LIN {X 0,Y 411.31,Z 349.876,A -85,B 0,C 180,E1 -10435.099,E2 -10435.099} C_VEL
LIN {X 0,Y 411.512,Z 349.85,A -85,B 0,C 180,E1 -10438.042,E2 -10438.042} C_VEL
LIN {X 0,Y 411.64,Z 349.837,A -85,B 0,C 180,E1 -10440,E2 -10440} C_VEL
LIN {X 0,Y 411.465,Z 349.857,A -85,B 0,C 180,E1 -10442.937,E2 -10442.937} C_VEL
LIN {X 0,Y 411.458,Z 349.857,A -85,B 0,C 180,E1 -10446.867,E2 -10446.867} C_VEL
LIN {X 0,Y 411.292,Z 349.877,A -85,B 0,C 180,E1 -10449.839,E2 -10449.839} C_VEL
LIN {X 0,Y 411.303,Z 349.874,A -85,B 0,C 180,E1 -10453.104,E2 -10453.104} C_VEL
LIN {X 0,Y 411.26,Z 349.883,A -85,B 0,C 180,E1 -10456.869,E2 -10456.869} C_VEL
LIN {X 0,Y 411.228,Z 349.888,A -85,B 0,C 180,E1 -10459.987,E2 -10459.987} C_VEL
LIN {X 0,Y 411.201,Z 349.893,A -85,B 0,C 180,E1 -10463.148,E2 -10463.148} C_VEL
LIN {X 0,Y 411.235,Z 349.889,A -85,B 0,C 180,E1 -10466.381,E2 -10466.381} C_VEL
LIN {X 0,Y 411.209,Z 349.89,A -85,B 0,C 180,E1 -10469.712,E2 -10469.712} C_VEL
LIN {X 0,Y 411.204,Z 349.89,A -85,B 0,C 180,E1 -10473.156,E2 -10473.156} C_VEL
LIN {X 0,Y 411.193,Z 349.891,A -85,B 0,C 180,E1 -10476.553,E2 -10476.553} C_VEL
LIN {X 0,Y 411.247,Z 349.991,A -85,B 0,C 180,E1 -10479.561,E2 -10479.561} C_VEL
LIN {X 0,Y 412.074,Z 354.924,A -85,B 0,C 180,E1 -10483.016,E2 -10483.016} C_VEL
LIN {X 0,Y 412.925,Z 360.046,A -85,B 0,C 180,E1 -10486.331,E2 -10486.331} C_VEL
LIN {X 0,Y 413.217,Z 363.579,A -85,B 0,C 180,E1 -10488.448,E2 -10488.448} C_VEL
LIN {X 0,Y 412.818,Z 369.165,A -85,B 0,C 180,E1 -10491.547,E2 -10491.547} C_VEL
LIN {X 0,Y 412.354,Z 375.474,A -85,B 0,C 180,E1 -10494.894,E2 -10494.894} C_VEL
LIN {X 0,Y 411.903,Z 382.668,A -85,B 0,C 180,E1 -10498.552,E2 -10498.552} C_VEL
LIN {X 0,Y 411.323,Z 389.578,A -85,B 0,C 180,E1 -10501.974,E2 -10501.974} C_VEL
LIN {X 0,Y 410.999,Z 395.754,A -85,B 0,C 180,E1 -10505.028,E2 -10505.028} C_VEL
LIN {X 0,Y 415.661,Z 413.767,A -85,B 0,C 180,E1 -10505.779,E2 -10505.779} C_VEL
LIN {X 0,Y 418.601,Z 427.932,A -85,B 0,C 180,E1 -10506.506,E2 -10506.506} C_VEL
LIN {X 0,Y 419.89,Z 436.709,A -85,B 0,C 180,E1 -10507.01,E2 -10507.01} C_VEL
LIN {X 0,Y 418.871,Z 450.945,A -85,B 0,C 180,E1 -10507.821,E2 -10507.821} C_VEL
LIN {X 0,Y 417.535,Z 464.473,A -85,B 0,C 180,E1 -10508.784,E2 -10508.784} C_VEL
LIN {X 0,Y 416.15,Z 478.262,A -85,B 0,C 180,E1 -10510.003,E2 -10510.003} C_VEL
LIN {X 0,Y 414.83,Z 490.734,A -85,B 0,C 180,E1 -10511.349,E2 -10511.349} C_VEL
LIN {X 0,Y 413.539,Z 503.017,A -85,B 0,C 180,E1 -10512.953,E2 -10512.953} C_VEL
LIN {X 0,Y 412.356,Z 513.929,A -85,B 0,C 180,E1 -10514.683,E2 -10514.683} C_VEL
LIN {X 0,Y 411.484,Z 523.109,A -85,B 0,C 180,E1 -10516.435,E2 -10516.435} C_VEL
LIN {X 0,Y 410.878,Z 530.585,A -85,B 0,C 180,E1 -10518.156,E2 -10518.156} C_VEL
LIN {X 0,Y 410.341,Z 537.64,A -85,B 0,C 180,E1 -10520.139,E2 -10520.139} C_VEL
LIN {X 0,Y 410.152,Z 543.2,A -85,B 0,C 180,E1 -10522.121,E2 -10522.121} C_VEL
LIN {X 0,Y 409.988,Z 547.402,A -85,B 0,C 180,E1 -10524.097,E2 -10524.097} C_VEL
LIN {X 0,Y 409.933,Z 550.351,A -85,B 0,C 180,E1 -10526.068,E2 -10526.068} C_VEL
LIN {X 0,Y 410.009,Z 552.115,A -85,B 0,C 180,E1 -10528.036,E2 -10528.036} C_VEL
LIN {X 0,Y 409.968,Z 552.715,A -85,B 0,C 180,E1 -10530,E2 -10530} C_VEL
LIN {X 0,Y 410.009,Z 552.11,A -85,B 0,C 180,E1 -10531.965,E2 -10531.965} C_VEL
LIN {X 0,Y 409.936,Z 550.342,A -85,B 0,C 180,E1 -10533.933,E2 -10533.933} C_VEL
LIN {X 0,Y 410.034,Z 547.395,A -85,B 0,C 180,E1 -10535.903,E2 -10535.903} C_VEL
LIN {X 0,Y 410.153,Z 543.193,A -85,B 0,C 180,E1 -10537.879,E2 -10537.879} C_VEL
LIN {X 0,Y 410.341,Z 537.627,A -85,B 0,C 180,E1 -10539.862,E2 -10539.862} C_VEL
LIN {X 0,Y 410.884,Z 530.561,A -85,B 0,C 180,E1 -10541.845,E2 -10541.845} C_VEL
LIN {X 0,Y 411.591,Z 521.772,A -85,B 0,C 180,E1 -10543.831,E2 -10543.831} C_VEL
LIN {X 0,Y 412.495,Z 512.449,A -85,B 0,C 180,E1 -10545.566,E2 -10545.566} C_VEL
LIN {X 0,Y 413.491,Z 502.979,A -85,B 0,C 180,E1 -10547.05,E2 -10547.05} C_VEL
LIN {X 0,Y 414.8,Z 491.133,A -85,B 0,C 180,E1 -10548.601,E2 -10548.601} C_VEL
LIN {X 0,Y 416.041,Z 479.441,A -85,B 0,C 180,E1 -10549.875,E2 -10549.875} C_VEL
LIN {X 0,Y 417.365,Z 465.924,A -85,B 0,C 180,E1 -10551.097,E2 -10551.097} C_VEL
LIN {X 0,Y 418.711,Z 452.668,A -85,B 0,C 180,E1 -10552.059,E2 -10552.059} C_VEL
LIN {X 0,Y 419.657,Z 439.382,A -85,B 0,C 180,E1 -10552.846,E2 -10552.846} C_VEL
LIN {X 0,Y 419.836,Z 435.502,A -85,B 0,C 180,E1 -10553.05,E2 -10553.05} C_VEL
LIN {X 0,Y 417.05,Z 420.044,A -85,B 0,C 180,E1 -10553.907,E2 -10553.907} C_VEL
LIN {X 0,Y 413.473,Z 405.19,A -85,B 0,C 180,E1 -10554.597,E2 -10554.597} C_VEL
LIN {X 0,Y 410.984,Z 395.734,A -85,B 0,C 180,E1 -10554.976,E2 -10554.976} C_VEL
LIN {X 0,Y 411.42,Z 388.428,A -85,B 0,C 180,E1 -10558.575,E2 -10558.575} C_VEL
LIN {X 0,Y 411.784,Z 382.677,A -85,B 0,C 180,E1 -10561.421,E2 -10561.421} C_VEL
LIN {X 0,Y 412.245,Z 377.131,A -85,B 0,C 180,E1 -10564.235,E2 -10564.235} C_VEL
LIN {X 0,Y 412.687,Z 370.278,A -85,B 0,C 180,E1 -10567.813,E2 -10567.813} C_VEL
LIN {X 0,Y 413.181,Z 364.609,A -85,B 0,C 180,E1 -10570.91,E2 -10570.91} C_VEL
LIN {X 0,Y 413.04,Z 361.111,A -85,B 0,C 180,E1 -10572.975,E2 -10572.975} C_VEL
LIN {X 0,Y 412.407,Z 356.805,A -85,B 0,C 180,E1 -10575.704,E2 -10575.704} C_VEL
LIN {X 0,Y 411.632,Z 352.375,A -85,B 0,C 180,E1 -10578.698,E2 -10578.698} C_VEL
LIN {X 0,Y 411.232,Z 349.887,A -85,B 0,C 180,E1 -10580.521,E2 -10580.521} C_VEL
LIN {X 0,Y 411.198,Z 349.896,A -85,B 0,C 180,E1 -10583.447,E2 -10583.447} C_VEL
LIN {X 0,Y 411.209,Z 349.891,A -85,B 0,C 180,E1 -10586.874,E2 -10586.874} C_VEL
LIN {X 0,Y 411.235,Z 349.888,A -85,B 0,C 180,E1 -10590.644,E2 -10590.644} C_VEL
LIN {X 0,Y 411.24,Z 349.887,A -85,B 0,C 180,E1 -10593.619,E2 -10593.619} C_VEL
LIN {X 0,Y 411.206,Z 349.892,A -85,B 0,C 180,E1 -10596.853,E2 -10596.853} C_VEL
LIN {X 0,Y 411.218,Z 349.89,A -85,B 0,C 180,E1 -10600.05,E2 -10600.05} C_VEL
LIN {X 0,Y 411.266,Z 349.885,A -85,B 0,C 180,E1 -10603.131,E2 -10603.131} C_VEL
LIN {X 0,Y 411.309,Z 349.878,A -85,B 0,C 180,E1 -10606.896,E2 -10606.896} C_VEL
LIN {X 0,Y 411.296,Z 349.879,A -85,B 0,C 180,E1 -10610.161,E2 -10610.161} C_VEL
LIN {X 0,Y 411.464,Z 349.857,A -85,B 0,C 180,E1 -10613.133,E2 -10613.133} C_VEL
LIN {X 0,Y 411.314,Z 349.878,A -85,B 0,C 180,E1 -10615.099,E2 -10615.099} C_VEL
LIN {X 0,Y 411.517,Z 349.851,A -85,B 0,C 180,E1 -10618.043,E2 -10618.043} C_VEL
LIN {X 0,Y 411.644,Z 349.834,A -85,B 0,C 180,E1 -10620,E2 -10620} C_VEL
LIN {X 0,Y 411.468,Z 349.855,A -85,B 0,C 180,E1 -10622.937,E2 -10622.937} C_VEL
LIN {X 0,Y 411.464,Z 349.853,A -85,B 0,C 180,E1 -10626.867,E2 -10626.867} C_VEL
LIN {X 0,Y 411.297,Z 349.876,A -85,B 0,C 180,E1 -10629.839,E2 -10629.839} C_VEL
LIN {X 0,Y 411.309,Z 349.855,A -85,B 0,C 180,E1 -10633.104,E2 -10633.104} C_VEL
LIN {X 0,Y 411.266,Z 349.881,A -85,B 0,C 180,E1 -10636.869,E2 -10636.869} C_VEL
LIN {X 0,Y 411.234,Z 349.867,A -85,B 0,C 180,E1 -10639.987,E2 -10639.987} C_VEL
LIN {X 0,Y 411.199,Z 349.888,A -85,B 0,C 180,E1 -10643.148,E2 -10643.148} C_VEL
LIN {X 0,Y 411.24,Z 349.874,A -85,B 0,C 180,E1 -10646.381,E2 -10646.381} C_VEL
LIN {X 0,Y 411.204,Z 349.887,A -85,B 0,C 180,E1 -10649.713,E2 -10649.713} C_VEL
LIN {X 0,Y 411.209,Z 349.879,A -85,B 0,C 180,E1 -10653.156,E2 -10653.156} C_VEL
LIN {X 0,Y 411.199,Z 349.892,A -85,B 0,C 180,E1 -10656.553,E2 -10656.553} C_VEL
LIN {X 0,Y 411.222,Z 349.888,A -85,B 0,C 180,E1 -10659.729,E2 -10659.729} C_VEL
LIN {X 0,Y 411.176,Z 349.894,A -85,B 0,C 180,E1 -10663.133,E2 -10663.133} C_VEL
LIN {X 0,Y 411.172,Z 349.897,A -85,B 0,C 180,E1 -10665.881,E2 -10665.881} C_VEL
LIN {X 0,Y 411.079,Z 349.91,A -85,B 0,C 180,E1 -10668.785,E2 -10668.785} C_VEL
LIN {X 0,Y 410.902,Z 349.929,A -85,B 0,C 180,E1 -10670.739,E2 -10670.739} C_VEL
LIN {X 0,Y 410.796,Z 350.166,A -85,B 0,C 180,E1 -10671.982,E2 -10671.982} C_VEL
LIN {X 0,Y 410.745,Z 352.725,A -85,B 0,C 180,E1 -10675.215,E2 -10675.215} C_VEL
LIN {X 0,Y 410.63,Z 355.755,A -85,B 0,C 180,E1 -10678.844,E2 -10678.844} C_VEL
LIN {X 0,Y 410.543,Z 357.94,A -85,B 0,C 180,E1 -10681.358,E2 -10681.358} C_VEL
LIN {X 0,Y 410.453,Z 361.284,A -85,B 0,C 180,E1 -10684.958,E2 -10684.958} C_VEL
LIN {X 0,Y 410.469,Z 361.411,A -85,B 0,C 180,E1 -10685.092,E2 -10685.092} C_VEL
LIN {X 0,Y 411.351,Z 364.267,A -85,B 0,C 180,E1 -10685.219,E2 -10685.219} C_VEL
LIN {X 0,Y 416.508,Z 378.808,A -85,B 0,C 180,E1 -10685.964,E2 -10685.964} C_VEL
LIN {X 0,Y 420.599,Z 392.516,A -85,B 0,C 180,E1 -10686.784,E2 -10686.784} C_VEL
LIN {X 0,Y 420.891,Z 395.97,A -85,B 0,C 180,E1 -10686.976,E2 -10686.976} C_VEL
LIN {X 0,Y 419.933,Z 410.109,A -85,B 0,C 180,E1 -10687.749,E2 -10687.749} C_VEL
LIN {X 0,Y 418.794,Z 424.059,A -85,B 0,C 180,E1 -10688.721,E2 -10688.721} C_VEL
LIN {X 0,Y 417.545,Z 436.805,A -85,B 0,C 180,E1 -10689.815,E2 -10689.815} C_VEL
LIN {X 0,Y 416.305,Z 448.773,A -85,B 0,C 180,E1 -10691.06,E2 -10691.06} C_VEL
LIN {X 0,Y 415.011,Z 460.345,A -85,B 0,C 180,E1 -10692.507,E2 -10692.507} C_VEL
LIN {X 0,Y 413.9,Z 470.241,A -85,B 0,C 180,E1 -10693.983,E2 -10693.983} C_VEL
LIN {X 0,Y 412.931,Z 478.771,A -85,B 0,C 180,E1 -10695.486,E2 -10695.486} C_VEL
LIN {X 0,Y 412.127,Z 486.852,A -85,B 0,C 180,E1 -10697.191,E2 -10697.191} C_VEL
LIN {X 0,Y 411.308,Z 494.567,A -85,B 0,C 180,E1 -10699.166,E2 -10699.166} C_VEL
LIN {X 0,Y 410.784,Z 500.701,A -85,B 0,C 180,E1 -10701.142,E2 -10701.142} C_VEL
LIN {X 0,Y 410.362,Z 505.997,A -85,B 0,C 180,E1 -10703.379,E2 -10703.379} C_VEL
LIN {X 0,Y 410.148,Z 508.905,A -85,B 0,C 180,E1 -10705.085,E2 -10705.085} C_VEL
LIN {X 0,Y 410.158,Z 511.191,A -85,B 0,C 180,E1 -10707.053,E2 -10707.053} C_VEL
LIN {X 0,Y 410.003,Z 512.367,A -85,B 0,C 180,E1 -10709.017,E2 -10709.017} C_VEL
LIN {X 0,Y 410.003,Z 512.383,A -85,B 0,C 180,E1 -10710.982,E2 -10710.982} C_VEL
LIN {X 0,Y 410.158,Z 511.271,A -85,B 0,C 180,E1 -10712.946,E2 -10712.946} C_VEL
LIN {X 0,Y 410.145,Z 509.047,A -85,B 0,C 180,E1 -10714.915,E2 -10714.915} C_VEL
LIN {X 0,Y 410.384,Z 505.637,A -85,B 0,C 180,E1 -10716.885,E2 -10716.885} C_VEL
LIN {X 0,Y 410.497,Z 504.262,A -85,B 0,C 180,E1 -10717.521,E2 -10717.521} C_VEL
LIN {X 0,Y 409.965,Z 502.472,A -85,B 0,C 180,E1 -10718.304,E2 -10718.304} C_VEL
LIN {X 0,Y 407.343,Z 499.365,A -85,B 0,C 180,E1 -10719.574,E2 -10719.574} C_VEL
LIN {X 0,Y 404.825,Z 495.813,A -85,B 0,C 180,E1 -10720.834,E2 -10720.834} C_VEL
LIN {X 0,Y 404.462,Z 493.252,A -85,B 0,C 180,E1 -10721.589,E2 -10721.589} C_VEL
LIN {X 0,Y 405.265,Z 486.259,A -85,B 0,C 180,E1 -10723.345,E2 -10723.345} C_VEL
LIN {X 0,Y 406.118,Z 478.157,A -85,B 0,C 180,E1 -10725.045,E2 -10725.045} C_VEL
LIN {X 0,Y 407.381,Z 468.063,A -85,B 0,C 180,E1 -10726.796,E2 -10726.796} C_VEL
LIN {X 0,Y 408.561,Z 457.735,A -85,B 0,C 180,E1 -10728.296,E2 -10728.296} C_VEL
LIN {X 0,Y 409.885,Z 446.49,A -85,B 0,C 180,E1 -10729.663,E2 -10729.663} C_VEL
LIN {X 0,Y 411.271,Z 434.248,A -85,B 0,C 180,E1 -10730.899,E2 -10730.899} C_VEL
LIN {X 0,Y 412.521,Z 420.866,A -85,B 0,C 180,E1 -10732.012,E2 -10732.012} C_VEL
LIN {X 0,Y 413.763,Z 405.942,A -85,B 0,C 180,E1 -10732.996,E2 -10732.996} C_VEL
LIN {X 0,Y 414.341,Z 396.576,A -85,B 0,C 180,E1 -10733.493,E2 -10733.493} C_VEL
LIN {X 0,Y 413.558,Z 392.314,A -85,B 0,C 180,E1 -10733.762,E2 -10733.762} C_VEL
LIN {X 0,Y 409.3,Z 378.287,A -85,B 0,C 180,E1 -10734.619,E2 -10734.619} C_VEL
LIN {X 0,Y 404.354,Z 364.726,A -85,B 0,C 180,E1 -10735.337,E2 -10735.337} C_VEL
LIN {X 0,Y 403.381,Z 361.733,A -85,B 0,C 180,E1 -10735.481,E2 -10735.481} C_VEL
LIN {X 0,Y 403.521,Z 358.376,A -85,B 0,C 180,E1 -10739.187,E2 -10739.187} C_VEL
LIN {X 0,Y 403.597,Z 355.417,A -85,B 0,C 180,E1 -10742.67,E2 -10742.67} C_VEL
LIN {X 0,Y 403.706,Z 353.423,A -85,B 0,C 180,E1 -10745.094,E2 -10745.094} C_VEL
LIN {X 0,Y 403.77,Z 350.819,A -85,B 0,C 180,E1 -10748.439,E2 -10748.439} C_VEL
LIN {X 0,Y 404.036,Z 350.78,A -85,B 0,C 180,E1 -10751.375,E2 -10751.375} C_VEL
LIN {X 0,Y 404.146,Z 350.769,A -85,B 0,C 180,E1 -10754.522,E2 -10754.522} C_VEL
LIN {X 0,Y 404.135,Z 350.77,A -85,B 0,C 180,E1 -10757.295,E2 -10757.295} C_VEL
LIN {X 0,Y 404.167,Z 350.765,A -85,B 0,C 180,E1 -10759.955,E2 -10759.955} C_VEL
LIN {X 0,Y 404.138,Z 350.768,A -85,B 0,C 180,E1 -10763.124,E2 -10763.124} C_VEL
LIN {X 0,Y 404.143,Z 350.763,A -85,B 0,C 180,E1 -10766.187,E2 -10766.187} C_VEL
LIN {X 0,Y 404.153,Z 350.769,A -85,B 0,C 180,E1 -10769.715,E2 -10769.715} C_VEL
LIN {X 0,Y 404.194,Z 350.75,A -85,B 0,C 180,E1 -10773.123,E2 -10773.123} C_VEL
LIN {X 0,Y 404.175,Z 350.762,A -85,B 0,C 180,E1 -10775.334,E2 -10775.334} C_VEL
LIN {X 0,Y 404.137,Z 350.759,A -85,B 0,C 180,E1 -10778.58,E2 -10778.58} C_VEL
LIN {X 0,Y 404.209,Z 350.756,A -85,B 0,C 180,E1 -10781.762,E2 -10781.762} C_VEL
LIN {X 0,Y 404.206,Z 350.756,A -85,B 0,C 180,E1 -10784.882,E2 -10784.882} C_VEL
LIN {X 0,Y 404.268,Z 350.74,A -85,B 0,C 180,E1 -10787.959,E2 -10787.959} C_VEL
LIN {X 0,Y 404.431,Z 350.731,A -85,B 0,C 180,E1 -10792.099,E2 -10792.099} C_VEL
LIN {X 0,Y 404.422,Z 350.735,A -85,B 0,C 180,E1 -10794.015,E2 -10794.015} C_VEL
LIN {X 0,Y 404.481,Z 350.726,A -85,B 0,C 180,E1 -10798.008,E2 -10798.008} C_VEL
LIN {X 0,Y 404.609,Z 350.713,A -85,B 0,C 180,E1 -10800,E2 -10800} C_VEL
LIN {X 0,Y 404.422,Z 350.734,A -85,B 0,C 180,E1 -10802.988,E2 -10802.988} C_VEL
LIN {X 0,Y 404.41,Z 350.735,A -85,B 0,C 180,E1 -10806.987,E2 -10806.987} C_VEL
LIN {X 0,Y 404.257,Z 350.753,A -85,B 0,C 180,E1 -10810.012,E2 -10810.012} C_VEL
LIN {X 0,Y 404.264,Z 350.751,A -85,B 0,C 180,E1 -10813.211,E2 -10813.211} C_VEL
LIN {X 0,Y 404.213,Z 350.762,A -85,B 0,C 180,E1 -10817.007,E2 -10817.007} C_VEL
LIN {X 0,Y 404.161,Z 350.765,A -85,B 0,C 180,E1 -10820.352,E2 -10820.352} C_VEL
LIN {X 0,Y 404.167,Z 350.767,A -85,B 0,C 180,E1 -10823.575,E2 -10823.575} C_VEL
LIN {X 0,Y 404.181,Z 350.766,A -85,B 0,C 180,E1 -10825.766,E2 -10825.766} C_VEL
LIN {X 0,Y 404.195,Z 350.764,A -85,B 0,C 180,E1 -10828,E2 -10828} C_VEL
LIN {X 0,Y 404.143,Z 350.769,A -85,B 0,C 180,E1 -10831.56,E2 -10831.56} C_VEL
LIN {X 0,Y 404.183,Z 350.765,A -85,B 0,C 180,E1 -10835.016,E2 -10835.016} C_VEL
LIN {X 0,Y 404.181,Z 350.764,A -85,B 0,C 180,E1 -10838.994,E2 -10838.994} C_VEL
LIN {X 0,Y 404.996,Z 355.684,A -85,B 0,C 180,E1 -10842.592,E2 -10842.592} C_VEL
LIN {X 0,Y 405.915,Z 361.091,A -85,B 0,C 180,E1 -10846.168,E2 -10846.168} C_VEL
LIN {X 0,Y 406.21,Z 364.197,A -85,B 0,C 180,E1 -10848.07,E2 -10848.07} C_VEL
LIN {X 0,Y 406.01,Z 367.844,A -85,B 0,C 180,E1 -10850.174,E2 -10850.174} C_VEL
LIN {X 0,Y 405.599,Z 372.688,A -85,B 0,C 180,E1 -10852.85,E2 -10852.85} C_VEL
LIN {X 0,Y 405.241,Z 378.02,A -85,B 0,C 180,E1 -10855.693,E2 -10855.693} C_VEL
LIN {X 0,Y 404.69,Z 384.782,A -85,B 0,C 180,E1 -10859.183,E2 -10859.183} C_VEL
LIN {X 0,Y 404.193,Z 391.265,A -85,B 0,C 180,E1 -10862.47,E2 -10862.47} C_VEL
LIN {X 0,Y 403.981,Z 395.421,A -85,B 0,C 180,E1 -10864.573,E2 -10864.573} C_VEL
LIN {X 0,Y 407.461,Z 408.511,A -85,B 0,C 180,E1 -10865.113,E2 -10865.113} C_VEL
LIN {X 0,Y 410.905,Z 423.49,A -85,B 0,C 180,E1 -10865.862,E2 -10865.862} C_VEL
LIN {X 0,Y 413.24,Z 437.616,A -85,B 0,C 180,E1 -10866.69,E2 -10866.69} C_VEL
LIN {X 0,Y 412.24,Z 450.889,A -85,B 0,C 180,E1 -10867.464,E2 -10867.464} C_VEL
LIN {X 0,Y 410.893,Z 464.128,A -85,B 0,C 180,E1 -10868.424,E2 -10868.424} C_VEL
LIN {X 0,Y 409.409,Z 477.913,A -85,B 0,C 180,E1 -10869.659,E2 -10869.659} C_VEL
LIN {X 0,Y 408.148,Z 489.327,A -85,B 0,C 180,E1 -10870.904,E2 -10870.904} C_VEL
LIN {X 0,Y 406.905,Z 500.891,A -85,B 0,C 180,E1 -10872.407,E2 -10872.407} C_VEL
LIN {X 0,Y 405.688,Z 510.624,A -85,B 0,C 180,E1 -10873.909,E2 -10873.909} C_VEL
LIN {X 0,Y 404.724,Z 520.201,A -85,B 0,C 180,E1 -10875.674,E2 -10875.674} C_VEL
LIN {X 0,Y 404.052,Z 528.192,A -85,B 0,C 180,E1 -10877.443,E2 -10877.443} C_VEL
LIN {X 0,Y 403.433,Z 535.655,A -85,B 0,C 180,E1 -10879.461,E2 -10879.461} C_VEL
LIN {X 0,Y 403.119,Z 541.586,A -85,B 0,C 180,E1 -10881.478,E2 -10881.478} C_VEL
LIN {X 0,Y 402.981,Z 545.114,A -85,B 0,C 180,E1 -10882.988,E2 -10882.988} C_VEL
LIN {X 0,Y 402.899,Z 548.682,A -85,B 0,C 180,E1 -10884.997,E2 -10884.997} C_VEL
LIN {X 0,Y 402.872,Z 551.03,A -85,B 0,C 180,E1 -10887.001,E2 -10887.001} C_VEL
LIN {X 0,Y 402.899,Z 552.213,A -85,B 0,C 180,E1 -10889.001,E2 -10889.001} C_VEL
LIN {X 0,Y 402.899,Z 552.212,A -85,B 0,C 180,E1 -10891,E2 -10891} C_VEL
LIN {X 0,Y 402.872,Z 551.023,A -85,B 0,C 180,E1 -10893,E2 -10893} C_VEL
LIN {X 0,Y 402.913,Z 548.672,A -85,B 0,C 180,E1 -10895.004,E2 -10895.004} C_VEL
LIN {X 0,Y 402.99,Z 545.106,A -85,B 0,C 180,E1 -10897.012,E2 -10897.012} C_VEL
LIN {X 0,Y 403.158,Z 540.237,A -85,B 0,C 180,E1 -10899.027,E2 -10899.027} C_VEL
LIN {X 0,Y 403.595,Z 533.943,A -85,B 0,C 180,E1 -10901.044,E2 -10901.044} C_VEL
LIN {X 0,Y 404.159,Z 526.042,A -85,B 0,C 180,E1 -10903.066,E2 -10903.066} C_VEL
LIN {X 0,Y 404.997,Z 517.655,A -85,B 0,C 180,E1 -10904.831,E2 -10904.831} C_VEL
LIN {X 0,Y 406.041,Z 507.558,A -85,B 0,C 180,E1 -10906.595,E2 -10906.595} C_VEL
LIN {X 0,Y 407.217,Z 497.246,A -85,B 0,C 180,E1 -10908.099,E2 -10908.099} C_VEL
LIN {X 0,Y 408.578,Z 484.967,A -85,B 0,C 180,E1 -10909.599,E2 -10909.599} C_VEL
LIN {X 0,Y 410.107,Z 471.312,A -85,B 0,C 180,E1 -10910.962,E2 -10910.962} C_VEL
LIN {X 0,Y 411.554,Z 457.634,A -85,B 0,C 180,E1 -10912.067,E2 -10912.067} C_VEL
LIN {X 0,Y 412.703,Z 444.208,A -85,B 0,C 180,E1 -10912.946,E2 -10912.946} C_VEL
LIN {X 0,Y 413.219,Z 436.929,A -85,B 0,C 180,E1 -10913.345,E2 -10913.345} C_VEL
LIN {X 0,Y 410.448,Z 421.063,A -85,B 0,C 180,E1 -10914.265,E2 -10914.265} C_VEL
LIN {X 0,Y 406.731,Z 405.838,A -85,B 0,C 180,E1 -10915.005,E2 -10915.005} C_VEL
LIN {X 0,Y 403.993,Z 395.364,A -85,B 0,C 180,E1 -10915.447,E2 -10915.447} C_VEL
LIN {X 0,Y 404.44,Z 388.099,A -85,B 0,C 180,E1 -10919.115,E2 -10919.115} C_VEL
LIN {X 0,Y 404.792,Z 382.987,A -85,B 0,C 180,E1 -10921.708,E2 -10921.708} C_VEL
LIN {X 0,Y 405.273,Z 376.841,A -85,B 0,C 180,E1 -10924.909,E2 -10924.909} C_VEL
LIN {X 0,Y 405.685,Z 371.125,A -85,B 0,C 180,E1 -10927.952,E2 -10927.952} C_VEL
LIN {X 0,Y 406.204,Z 365.51,A -85,B 0,C 180,E1 -10931.107,E2 -10931.107} C_VEL
LIN {X 0,Y 405.994,Z 361.772,A -85,B 0,C 180,E1 -10933.361,E2 -10933.361} C_VEL
LIN {X 0,Y 405.333,Z 357.583,A -85,B 0,C 180,E1 -10936.088,E2 -10936.088} C_VEL
LIN {X 0,Y 404.697,Z 353.786,A -85,B 0,C 180,E1 -10938.707,E2 -10938.707} C_VEL
LIN {X 0,Y 404.172,Z 350.77,A -85,B 0,C 180,E1 -10941.085,E2 -10941.085} C_VEL
LIN {X 0,Y 404.188,Z 350.769,A -85,B 0,C 180,E1 -10944.984,E2 -10944.984} C_VEL
LIN {X 0,Y 404.144,Z 350.769,A -85,B 0,C 180,E1 -10948.554,E2 -10948.554} C_VEL
LIN {X 0,Y 404.198,Z 350.763,A -85,B 0,C 180,E1 -10952.001,E2 -10952.001} C_VEL
LIN {X 0,Y 404.18,Z 350.766,A -85,B 0,C 180,E1 -10955.335,E2 -10955.335} C_VEL
LIN {X 0,Y 404.142,Z 350.771,A -85,B 0,C 180,E1 -10958.581,E2 -10958.581} C_VEL
LIN {X 0,Y 404.213,Z 350.762,A -85,B 0,C 180,E1 -10961.762,E2 -10961.762} C_VEL
LIN {X 0,Y 404.21,Z 350.764,A -85,B 0,C 180,E1 -10964.882,E2 -10964.882} C_VEL
LIN {X 0,Y 404.26,Z 350.757,A -85,B 0,C 180,E1 -10967.959,E2 -10967.959} C_VEL
LIN {X 0,Y 404.437,Z 350.736,A -85,B 0,C 180,E1 -10972.1,E2 -10972.1} C_VEL
LIN {X 0,Y 404.427,Z 350.734,A -85,B 0,C 180,E1 -10974.015,E2 -10974.015} C_VEL
LIN {X 0,Y 404.486,Z 350.726,A -85,B 0,C 180,E1 -10978.009,E2 -10978.009} C_VEL
LIN {X 0,Y 404.613,Z 350.709,A -85,B 0,C 180,E1 -10980,E2 -10980} C_VEL
LIN {X 0,Y 404.425,Z 350.732,A -85,B 0,C 180,E1 -10982.988,E2 -10982.988} C_VEL
LIN {X 0,Y 404.416,Z 350.731,A -85,B 0,C 180,E1 -10986.987,E2 -10986.987} C_VEL
LIN {X 0,Y 404.262,Z 350.753,A -85,B 0,C 180,E1 -10990.012,E2 -10990.012} C_VEL
LIN {X 0,Y 404.27,Z 350.732,A -85,B 0,C 180,E1 -10993.211,E2 -10993.211} C_VEL
LIN {X 0,Y 404.219,Z 350.758,A -85,B 0,C 180,E1 -10997.007,E2 -10997.007} C_VEL
LIN {X 0,Y 404.167,Z 350.745,A -85,B 0,C 180,E1 -11000.352,E2 -11000.352} C_VEL
LIN {X 0,Y 404.166,Z 350.764,A -85,B 0,C 180,E1 -11003.575,E2 -11003.575} C_VEL
LIN {X 0,Y 404.186,Z 350.757,A -85,B 0,C 180,E1 -11005.766,E2 -11005.766} C_VEL
LIN {X 0,Y 404.198,Z 350.751,A -85,B 0,C 180,E1 -11008,E2 -11008} C_VEL
LIN {X 0,Y 404.142,Z 350.769,A -85,B 0,C 180,E1 -11011.558,E2 -11011.558} C_VEL
LIN {X 0,Y 404.189,Z 350.761,A -85,B 0,C 180,E1 -11015.016,E2 -11015.016} C_VEL
LIN {X 0,Y 404.162,Z 350.766,A -85,B 0,C 180,E1 -11018.756,E2 -11018.756} C_VEL
LIN {X 0,Y 404.126,Z 350.771,A -85,B 0,C 180,E1 -11021.6,E2 -11021.6} C_VEL
LIN {X 0,Y 404.149,Z 350.77,A -85,B 0,C 180,E1 -11024.522,E2 -11024.522} C_VEL
LIN {X 0,Y 404.109,Z 350.778,A -85,B 0,C 180,E1 -11027.291,E2 -11027.291} C_VEL
LIN {X 0,Y 403.964,Z 350.794,A -85,B 0,C 180,E1 -11029.951,E2 -11029.951} C_VEL
LIN {X 0,Y 403.774,Z 350.818,A -85,B 0,C 180,E1 -11031.56,E2 -11031.56} C_VEL
LIN {X 0,Y 403.713,Z 353.359,A -85,B 0,C 180,E1 -11034.937,E2 -11034.937} C_VEL
LIN {X 0,Y 403.601,Z 356.354,A -85,B 0,C 180,E1 -11038.567,E2 -11038.567} C_VEL
LIN {X 0,Y 403.474,Z 359.269,A -85,B 0,C 180,E1 -11041.945,E2 -11041.945} C_VEL
LIN {X 0,Y 403.403,Z 361.781,A -85,B 0,C 180,E1 -11044.628,E2 -11044.628} C_VEL
LIN {X 0,Y 404.279,Z 364.641,A -85,B 0,C 180,E1 -11044.754,E2 -11044.754} C_VEL
LIN {X 0,Y 409.095,Z 377.723,A -85,B 0,C 180,E1 -11045.444,E2 -11045.444} C_VEL
LIN {X 0,Y 413.466,Z 392.008,A -85,B 0,C 180,E1 -11046.313,E2 -11046.313} C_VEL
LIN {X 0,Y 414.375,Z 395.533,A -85,B 0,C 180,E1 -11046.552,E2 -11046.552} C_VEL
LIN {X 0,Y 413.532,Z 408.489,A -85,B 0,C 180,E1 -11047.254,E2 -11047.254} C_VEL
LIN {X 0,Y 412.317,Z 422.841,A -85,B 0,C 180,E1 -11048.239,E2 -11048.239} C_VEL
LIN {X 0,Y 411.026,Z 435.875,A -85,B 0,C 180,E1 -11049.349,E2 -11049.349} C_VEL
LIN {X 0,Y 409.819,Z 447.004,A -85,B 0,C 180,E1 -11050.489,E2 -11050.489} C_VEL
LIN {X 0,Y 408.429,Z 458.929,A -85,B 0,C 180,E1 -11051.956,E2 -11051.956} C_VEL
LIN {X 0,Y 407.207,Z 469.072,A -85,B 0,C 180,E1 -11053.454,E2 -11053.454} C_VEL
LIN {X 0,Y 406.053,Z 478.989,A -85,B 0,C 180,E1 -11055.209,E2 -11055.209} C_VEL
LIN {X 0,Y 405.187,Z 487.203,A -85,B 0,C 180,E1 -11056.968,E2 -11056.968} C_VEL
LIN {X 0,Y 404.299,Z 494.918,A -85,B 0,C 180,E1 -11058.976,E2 -11058.976} C_VEL
LIN {X 0,Y 403.745,Z 501.051,A -85,B 0,C 180,E1 -11060.986,E2 -11060.986} C_VEL
LIN {X 0,Y 403.345,Z 505.785,A -85,B 0,C 180,E1 -11062.994,E2 -11062.994} C_VEL
LIN {X 0,Y 403.088,Z 509.253,A -85,B 0,C 180,E1 -11064.998,E2 -11064.998} C_VEL
LIN {X 0,Y 403.094,Z 511.538,A -85,B 0,C 180,E1 -11067.001,E2 -11067.001} C_VEL
LIN {X 0,Y 402.927,Z 512.714,A -85,B 0,C 180,E1 -11069,E2 -11069} C_VEL
LIN {X 0,Y 402.927,Z 512.73,A -85,B 0,C 180,E1 -11070.999,E2 -11070.999} C_VEL
LIN {X 0,Y 403.093,Z 511.617,A -85,B 0,C 180,E1 -11072.998,E2 -11072.998} C_VEL
LIN {X 0,Y 403.085,Z 509.393,A -85,B 0,C 180,E1 -11075.001,E2 -11075.001} C_VEL
LIN {X 0,Y 403.341,Z 505.983,A -85,B 0,C 180,E1 -11077.005,E2 -11077.005} C_VEL
LIN {X 0,Y 403.729,Z 501.313,A -85,B 0,C 180,E1 -11079.013,E2 -11079.013} C_VEL
LIN {X 0,Y 404.264,Z 495.26,A -85,B 0,C 180,E1 -11081.024,E2 -11081.024} C_VEL
LIN {X 0,Y 404.462,Z 493.252,A -85,B 0,C 180,E1 -11081.589,E2 -11081.589} C_VEL
LIN {X 0,Y 404.128,Z 490.58,A -85,B 0,C 180,E1 -11082.334,E2 -11082.334} C_VEL
LIN {X 0,Y 401.797,Z 486.107,A -85,B 0,C 180,E1 -11083.55,E2 -11083.55} C_VEL
LIN {X 0,Y 399.55,Z 481.216,A -85,B 0,C 180,E1 -11084.742,E2 -11084.742} C_VEL
LIN {X 0,Y 399.344,Z 477.83,A -85,B 0,C 180,E1 -11085.437,E2 -11085.437} C_VEL
LIN {X 0,Y 400.579,Z 468.409,A -85,B 0,C 180,E1 -11087.089,E2 -11087.089} C_VEL
LIN {X 0,Y 401.815,Z 458.178,A -85,B 0,C 180,E1 -11088.601,E2 -11088.601} C_VEL
LIN {X 0,Y 403.174,Z 447.173,A -85,B 0,C 180,E1 -11089.964,E2 -11089.964} C_VEL
LIN {X 0,Y 404.647,Z 434.591,A -85,B 0,C 180,E1 -11091.257,E2 -11091.257} C_VEL
LIN {X 0,Y 405.96,Z 421.208,A -85,B 0,C 180,E1 -11092.387,E2 -11092.387} C_VEL
LIN {X 0,Y 407.247,Z 406.282,A -85,B 0,C 180,E1 -11093.385,E2 -11093.385} C_VEL
LIN {X 0,Y 407.775,Z 398.075,A -85,B 0,C 180,E1 -11093.834,E2 -11093.834} C_VEL
LIN {X 0,Y 406.182,Z 390.883,A -85,B 0,C 180,E1 -11094.307,E2 -11094.307} C_VEL
LIN {X 0,Y 401.522,Z 376.103,A -85,B 0,C 180,E1 -11095.219,E2 -11095.219} C_VEL
LIN {X 0,Y 396.412,Z 362.661,A -85,B 0,C 180,E1 -11095.94,E2 -11095.94} C_VEL
LIN {X 0,Y 396.348,Z 362.069,A -85,B 0,C 180,E1 -11095.992,E2 -11095.992} C_VEL
LIN {X 0,Y 396.472,Z 358.768,A -85,B 0,C 180,E1 -11099.704,E2 -11099.704} C_VEL
LIN {X 0,Y 396.533,Z 356.737,A -85,B 0,C 180,E1 -11102.12,E2 -11102.12} C_VEL
LIN {X 0,Y 396.651,Z 353.744,A -85,B 0,C 180,E1 -11105.782,E2 -11105.782} C_VEL
LIN {X 0,Y 396.715,Z 351.798,A -85,B 0,C 180,E1 -11108.319,E2 -11108.319} C_VEL
LIN {X 0,Y 396.942,Z 351.664,A -85,B 0,C 180,E1 -11110.926,E2 -11110.926} C_VEL
LIN {X 0,Y 397.096,Z 351.644,A -85,B 0,C 180,E1 -11113.649,E2 -11113.649} C_VEL
LIN {X 0,Y 397.101,Z 351.646,A -85,B 0,C 180,E1 -11116.52,E2 -11116.52} C_VEL
LIN {X 0,Y 397.113,Z 351.646,A -85,B 0,C 180,E1 -11120.423,E2 -11120.423} C_VEL
LIN {X 0,Y 397.108,Z 351.645,A -85,B 0,C 180,E1 -11124.265,E2 -11124.265} C_VEL
LIN {X 0,Y 397.113,Z 351.634,A -85,B 0,C 180,E1 -11126.727,E2 -11126.727} C_VEL
LIN {X 0,Y 397.132,Z 351.641,A -85,B 0,C 180,E1 -11130.296,E2 -11130.296} C_VEL
LIN {X 0,Y 397.193,Z 351.622,A -85,B 0,C 180,E1 -11132.61,E2 -11132.61} C_VEL
LIN {X 0,Y 397.131,Z 351.644,A -85,B 0,C 180,E1 -11135.982,E2 -11135.982} C_VEL
LIN {X 0,Y 397.136,Z 351.623,A -85,B 0,C 180,E1 -11139.704,E2 -11139.704} C_VEL
LIN {X 0,Y 397.18,Z 351.635,A -85,B 0,C 180,E1 -11142.845,E2 -11142.845} C_VEL
LIN {X 0,Y 397.224,Z 351.612,A -85,B 0,C 180,E1 -11146.679,E2 -11146.679} C_VEL
LIN {X 0,Y 397.227,Z 351.631,A -85,B 0,C 180,E1 -11149.809,E2 -11149.809} C_VEL
LIN {X 0,Y 397.362,Z 351.614,A -85,B 0,C 180,E1 -11152.888,E2 -11152.888} C_VEL
LIN {X 0,Y 397.254,Z 351.626,A -85,B 0,C 180,E1 -11154.925,E2 -11154.925} C_VEL
LIN {X 0,Y 397.45,Z 351.602,A -85,B 0,C 180,E1 -11157.973,E2 -11157.973} C_VEL
LIN {X 0,Y 397.579,Z 351.589,A -85,B 0,C 180,E1 -11160,E2 -11160} C_VEL
LIN {X 0,Y 397.38,Z 351.612,A -85,B 0,C 180,E1 -11163.041,E2 -11163.041} C_VEL
LIN {X 0,Y 397.362,Z 351.613,A -85,B 0,C 180,E1 -11167.112,E2 -11167.112} C_VEL
LIN {X 0,Y 397.217,Z 351.63,A -85,B 0,C 180,E1 -11170.191,E2 -11170.191} C_VEL
LIN {X 0,Y 397.224,Z 351.628,A -85,B 0,C 180,E1 -11173.321,E2 -11173.321} C_VEL
LIN {X 0,Y 397.179,Z 351.636,A -85,B 0,C 180,E1 -11177.155,E2 -11177.155} C_VEL
LIN {X 0,Y 397.1,Z 351.644,A -85,B 0,C 180,E1 -11180.73,E2 -11180.73} C_VEL
LIN {X 0,Y 397.131,Z 351.644,A -85,B 0,C 180,E1 -11184.018,E2 -11184.018} C_VEL
LIN {X 0,Y 397.192,Z 351.638,A -85,B 0,C 180,E1 -11187.39,E2 -11187.39} C_VEL
LIN {X 0,Y 397.084,Z 351.65,A -85,B 0,C 180,E1 -11190.882,E2 -11190.882} C_VEL
LIN {X 0,Y 397.124,Z 351.645,A -85,B 0,C 180,E1 -11194.493,E2 -11194.493} C_VEL
LIN {X 0,Y 397.104,Z 351.647,A -85,B 0,C 180,E1 -11198.275,E2 -11198.275} C_VEL
LIN {X 0,Y 397.178,Z 352.022,A -85,B 0,C 180,E1 -11198.871,E2 -11198.871} C_VEL
LIN {X 0,Y 397.932,Z 356.448,A -85,B 0,C 180,E1 -11202.154,E2 -11202.154} C_VEL
LIN {X 0,Y 398.691,Z 360.851,A -85,B 0,C 180,E1 -11205.162,E2 -11205.162} C_VEL
LIN {X 0,Y 399.185,Z 364.804,A -85,B 0,C 180,E1 -11207.684,E2 -11207.684} C_VEL
LIN {X 0,Y 399.036,Z 368.711,A -85,B 0,C 180,E1 -11209.996,E2 -11209.996} C_VEL
LIN {X 0,Y 398.533,Z 374.33,A -85,B 0,C 180,E1 -11213.161,E2 -11213.161} C_VEL
LIN {X 0,Y 398.12,Z 379.701,A -85,B 0,C 180,E1 -11216.067,E2 -11216.067} C_VEL
LIN {X 0,Y 397.639,Z 385.576,A -85,B 0,C 180,E1 -11219.166,E2 -11219.166} C_VEL
LIN {X 0,Y 397.122,Z 392.182,A -85,B 0,C 180,E1 -11222.605,E2 -11222.605} C_VEL
LIN {X 0,Y 396.979,Z 395.051,A -85,B 0,C 180,E1 -11224.082,E2 -11224.082} C_VEL
LIN {X 0,Y 401.722,Z 412.862,A -85,B 0,C 180,E1 -11224.875,E2 -11224.875} C_VEL
LIN {X 0,Y 404.885,Z 427.748,A -85,B 0,C 180,E1 -11225.684,E2 -11225.684} C_VEL
LIN {X 0,Y 406.531,Z 439.554,A -85,B 0,C 180,E1 -11226.418,E2 -11226.418} C_VEL
LIN {X 0,Y 405.284,Z 454.213,A -85,B 0,C 180,E1 -11227.333,E2 -11227.333} C_VEL
LIN {X 0,Y 403.766,Z 468.168,A -85,B 0,C 180,E1 -11228.426,E2 -11228.426} C_VEL
LIN {X 0,Y 402.25,Z 481.149,A -85,B 0,C 180,E1 -11229.681,E2 -11229.681} C_VEL
LIN {X 0,Y 400.95,Z 492.746,A -85,B 0,C 180,E1 -11231.038,E2 -11231.038} C_VEL
LIN {X 0,Y 399.617,Z 503.963,A -85,B 0,C 180,E1 -11232.604,E2 -11232.604} C_VEL
LIN {X 0,Y 398.34,Z 514.597,A -85,B 0,C 180,E1 -11234.392,E2 -11234.392} C_VEL
LIN {X 0,Y 397.394,Z 523.459,A -85,B 0,C 180,E1 -11236.188,E2 -11236.188} C_VEL
LIN {X 0,Y 396.85,Z 529.885,A -85,B 0,C 180,E1 -11237.731,E2 -11237.731} C_VEL
LIN {X 0,Y 396.229,Z 536.94,A -85,B 0,C 180,E1 -11239.784,E2 -11239.784} C_VEL
LIN {X 0,Y 395.98,Z 542.5,A -85,B 0,C 180,E1 -11241.838,E2 -11241.838} C_VEL
LIN {X 0,Y 395.859,Z 546.707,A -85,B 0,C 180,E1 -11243.886,E2 -11243.886} C_VEL
LIN {X 0,Y 395.772,Z 549.656,A -85,B 0,C 180,E1 -11245.927,E2 -11245.927} C_VEL
LIN {X 0,Y 395.867,Z 551.421,A -85,B 0,C 180,E1 -11247.966,E2 -11247.966} C_VEL
LIN {X 0,Y 395.816,Z 552.022,A -85,B 0,C 180,E1 -11250,E2 -11250} C_VEL
LIN {X 0,Y 395.867,Z 551.417,A -85,B 0,C 180,E1 -11252.035,E2 -11252.035} C_VEL
LIN {X 0,Y 395.776,Z 549.645,A -85,B 0,C 180,E1 -11254.074,E2 -11254.074} C_VEL
LIN {X 0,Y 395.907,Z 546.488,A -85,B 0,C 180,E1 -11256.232,E2 -11256.232} C_VEL
LIN {X 0,Y 395.981,Z 542.49,A -85,B 0,C 180,E1 -11258.163,E2 -11258.163} C_VEL
LIN {X 0,Y 396.229,Z 536.922,A -85,B 0,C 180,E1 -11260.217,E2 -11260.217} C_VEL
LIN {X 0,Y 396.858,Z 529.855,A -85,B 0,C 180,E1 -11262.27,E2 -11262.27} C_VEL
LIN {X 0,Y 397.515,Z 522.294,A -85,B 0,C 180,E1 -11264.07,E2 -11264.07} C_VEL
LIN {X 0,Y 398.493,Z 513.194,A -85,B 0,C 180,E1 -11265.865,E2 -11265.865} C_VEL
LIN {X 0,Y 399.813,Z 502.272,A -85,B 0,C 180,E1 -11267.652,E2 -11267.652} C_VEL
LIN {X 0,Y 401.099,Z 490.872,A -85,B 0,C 180,E1 -11269.202,E2 -11269.202} C_VEL
LIN {X 0,Y 402.546,Z 478.73,A -85,B 0,C 180,E1 -11270.571,E2 -11270.571} C_VEL
LIN {X 0,Y 404.075,Z 465.217,A -85,B 0,C 180,E1 -11271.825,E2 -11271.825} C_VEL
LIN {X 0,Y 405.611,Z 450.941,A -85,B 0,C 180,E1 -11272.888,E2 -11272.888} C_VEL
LIN {X 0,Y 406.567,Z 438.628,A -85,B 0,C 180,E1 -11273.628,E2 -11273.628} C_VEL
LIN {X 0,Y 404.136,Z 423.742,A -85,B 0,C 180,E1 -11274.534,E2 -11274.534} C_VEL
LIN {X 0,Y 400.727,Z 409.073,A -85,B 0,C 180,E1 -11275.298,E2 -11275.298} C_VEL
LIN {X 0,Y 396.965,Z 395.052,A -85,B 0,C 180,E1 -11275.909,E2 -11275.909} C_VEL
LIN {X 0,Y 397.502,Z 387.769,A -85,B 0,C 180,E1 -11279.674,E2 -11279.674} C_VEL
LIN {X 0,Y 398,Z 381.044,A -85,B 0,C 180,E1 -11283.19,E2 -11283.19} C_VEL
LIN {X 0,Y 398.435,Z 375.352,A -85,B 0,C 180,E1 -11286.251,E2 -11286.251} C_VEL
LIN {X 0,Y 399.014,Z 368.622,A -85,B 0,C 180,E1 -11290.008,E2 -11290.008} C_VEL
LIN {X 0,Y 399.179,Z 364.723,A -85,B 0,C 180,E1 -11292.315,E2 -11292.315} C_VEL
LIN {X 0,Y 398.609,Z 360.308,A -85,B 0,C 180,E1 -11295.15,E2 -11295.15} C_VEL
LIN {X 0,Y 397.927,Z 356.365,A -85,B 0,C 180,E1 -11297.884,E2 -11297.884} C_VEL
LIN {X 0,Y 397.133,Z 351.645,A -85,B 0,C 180,E1 -11301.428,E2 -11301.428} C_VEL
LIN {X 0,Y 397.122,Z 351.647,A -85,B 0,C 180,E1 -11304.497,E2 -11304.497} C_VEL
LIN {X 0,Y 397.081,Z 351.65,A -85,B 0,C 180,E1 -11307.929,E2 -11307.929} C_VEL
LIN {X 0,Y 397.124,Z 351.643,A -85,B 0,C 180,E1 -11311.457,E2 -11311.457} C_VEL
LIN {X 0,Y 397.155,Z 351.64,A -85,B 0,C 180,E1 -11314.488,E2 -11314.488} C_VEL
LIN {X 0,Y 397.112,Z 351.647,A -85,B 0,C 180,E1 -11317.086,E2 -11317.086} C_VEL
LIN {X 0,Y 397.151,Z 351.64,A -85,B 0,C 180,E1 -11320.353,E2 -11320.353} C_VEL
LIN {X 0,Y 397.17,Z 351.639,A -85,B 0,C 180,E1 -11323.553,E2 -11323.553} C_VEL
LIN {X 0,Y 397.232,Z 351.632,A -85,B 0,C 180,E1 -11326.703,E2 -11326.703} C_VEL
LIN {X 0,Y 397.221,Z 351.633,A -85,B 0,C 180,E1 -11329.809,E2 -11329.809} C_VEL
LIN {X 0,Y 397.367,Z 351.613,A -85,B 0,C 180,E1 -11332.888,E2 -11332.888} C_VEL
LIN {X 0,Y 397.258,Z 351.627,A -85,B 0,C 180,E1 -11334.925,E2 -11334.925} C_VEL
LIN {X 0,Y 397.455,Z 351.602,A -85,B 0,C 180,E1 -11337.973,E2 -11337.973} C_VEL
LIN {X 0,Y 397.582,Z 351.585,A -85,B 0,C 180,E1 -11340,E2 -11340} C_VEL
LIN {X 0,Y 397.384,Z 351.608,A -85,B 0,C 180,E1 -11343.041,E2 -11343.041} C_VEL
LIN {X 0,Y 397.368,Z 351.609,A -85,B 0,C 180,E1 -11347.112,E2 -11347.112} C_VEL
LIN {X 0,Y 397.222,Z 351.63,A -85,B 0,C 180,E1 -11350.191,E2 -11350.191} C_VEL
LIN {X 0,Y 397.23,Z 351.609,A -85,B 0,C 180,E1 -11353.321,E2 -11353.321} C_VEL
LIN {X 0,Y 397.185,Z 351.634,A -85,B 0,C 180,E1 -11357.155,E2 -11357.155} C_VEL
LIN {X 0,Y 397.106,Z 351.625,A -85,B 0,C 180,E1 -11360.73,E2 -11360.73} C_VEL
LIN {X 0,Y 397.131,Z 351.643,A -85,B 0,C 180,E1 -11364.018,E2 -11364.018} C_VEL
LIN {X 0,Y 397.197,Z 351.619,A -85,B 0,C 180,E1 -11367.39,E2 -11367.39} C_VEL
LIN {X 0,Y 397.082,Z 351.647,A -85,B 0,C 180,E1 -11370.882,E2 -11370.882} C_VEL
LIN {X 0,Y 397.129,Z 351.635,A -85,B 0,C 180,E1 -11374.493,E2 -11374.493} C_VEL
LIN {X 0,Y 397.11,Z 351.645,A -85,B 0,C 180,E1 -11378.274,E2 -11378.274} C_VEL
LIN {X 0,Y 397.092,Z 351.649,A -85,B 0,C 180,E1 -11380.908,E2 -11380.908} C_VEL
LIN {X 0,Y 397.104,Z 351.648,A -85,B 0,C 180,E1 -11383.648,E2 -11383.648} C_VEL
LIN {X 0,Y 397.098,Z 351.65,A -85,B 0,C 180,E1 -11386.522,E2 -11386.522} C_VEL
LIN {X 0,Y 396.944,Z 351.669,A -85,B 0,C 180,E1 -11389.581,E2 -11389.581} C_VEL
LIN {X 0,Y 396.711,Z 351.706,A -85,B 0,C 180,E1 -11391.68,E2 -11391.68} C_VEL
LIN {X 0,Y 396.66,Z 353.949,A -85,B 0,C 180,E1 -11394.59,E2 -11394.59} C_VEL
LIN {X 0,Y 396.564,Z 356.95,A -85,B 0,C 180,E1 -11398.285,E2 -11398.285} C_VEL
LIN {X 0,Y 396.444,Z 359.612,A -85,B 0,C 180,E1 -11401.403,E2 -11401.403} C_VEL
LIN {X 0,Y 396.383,Z 362.24,A -85,B 0,C 180,E1 -11404.148,E2 -11404.148} C_VEL
LIN {X 0,Y 397.314,Z 365.115,A -85,B 0,C 180,E1 -11404.281,E2 -11404.281} C_VEL
LIN {X 0,Y 402.349,Z 378.653,A -85,B 0,C 180,E1 -11405.025,E2 -11405.025} C_VEL
LIN {X 0,Y 406.33,Z 391.682,A -85,B 0,C 180,E1 -11405.836,E2 -11405.836} C_VEL
LIN {X 0,Y 407.824,Z 397.904,A -85,B 0,C 180,E1 -11406.257,E2 -11406.257} C_VEL
LIN {X 0,Y 406.862,Z 410.818,A -85,B 0,C 180,E1 -11406.994,E2 -11406.994} C_VEL
LIN {X 0,Y 405.602,Z 424.767,A -85,B 0,C 180,E1 -11407.994,E2 -11407.994} C_VEL
LIN {X 0,Y 404.254,Z 437.51,A -85,B 0,C 180,E1 -11409.121,E2 -11409.121} C_VEL
LIN {X 0,Y 402.847,Z 449.492,A -85,B 0,C 180,E1 -11410.403,E2 -11410.403} C_VEL
LIN {X 0,Y 401.465,Z 461.049,A -85,B 0,C 180,E1 -11411.896,E2 -11411.896} C_VEL
LIN {X 0,Y 400.212,Z 470.946,A -85,B 0,C 180,E1 -11413.419,E2 -11413.419} C_VEL
LIN {X 0,Y 398.999,Z 480.602,A -85,B 0,C 180,E1 -11415.202,E2 -11415.202} C_VEL
LIN {X 0,Y 398.164,Z 488.636,A -85,B 0,C 180,E1 -11416.994,E2 -11416.994} C_VEL
LIN {X 0,Y 397.299,Z 495.27,A -85,B 0,C 180,E1 -11418.779,E2 -11418.779} C_VEL
LIN {X 0,Y 396.726,Z 501.401,A -85,B 0,C 180,E1 -11420.825,E2 -11420.825} C_VEL
LIN {X 0,Y 396.297,Z 506.134,A -85,B 0,C 180,E1 -11422.869,E2 -11422.869} C_VEL
LIN {X 0,Y 396.029,Z 509.601,A -85,B 0,C 180,E1 -11424.909,E2 -11424.909} C_VEL
LIN {X 0,Y 396.011,Z 511.886,A -85,B 0,C 180,E1 -11426.948,E2 -11426.948} C_VEL
LIN {X 0,Y 395.854,Z 513.061,A -85,B 0,C 180,E1 -11428.982,E2 -11428.982} C_VEL
LIN {X 0,Y 395.854,Z 513.077,A -85,B 0,C 180,E1 -11431.017,E2 -11431.017} C_VEL
LIN {X 0,Y 396.01,Z 511.964,A -85,B 0,C 180,E1 -11433.051,E2 -11433.051} C_VEL
LIN {X 0,Y 396.027,Z 509.74,A -85,B 0,C 180,E1 -11435.09,E2 -11435.09} C_VEL
LIN {X 0,Y 396.293,Z 506.33,A -85,B 0,C 180,E1 -11437.131,E2 -11437.131} C_VEL
LIN {X 0,Y 396.712,Z 501.66,A -85,B 0,C 180,E1 -11439.174,E2 -11439.174} C_VEL
LIN {X 0,Y 397.264,Z 495.608,A -85,B 0,C 180,E1 -11441.221,E2 -11441.221} C_VEL
LIN {X 0,Y 398.202,Z 487.973,A -85,B 0,C 180,E1 -11443.264,E2 -11443.264} C_VEL
LIN {X 0,Y 399.089,Z 479.834,A -85,B 0,C 180,E1 -11445.055,E2 -11445.055} C_VEL
LIN {X 0,Y 399.344,Z 477.83,A -85,B 0,C 180,E1 -11445.437,E2 -11445.437} C_VEL
LIN {X 0,Y 399.186,Z 474.34,A -85,B 0,C 180,E1 -11446.121,E2 -11446.121} C_VEL
LIN {X 0,Y 397.188,Z 468.6,A -85,B 0,C 180,E1 -11447.253,E2 -11447.253} C_VEL
LIN {X 0,Y 395.221,Z 462.47,A -85,B 0,C 180,E1 -11448.346,E2 -11448.346} C_VEL
LIN {X 0,Y 395.099,Z 458.325,A -85,B 0,C 180,E1 -11448.957,E2 -11448.957} C_VEL
LIN {X 0,Y 396.655,Z 446.243,A -85,B 0,C 180,E1 -11450.456,E2 -11450.456} C_VEL
LIN {X 0,Y 398.185,Z 433.535,A -85,B 0,C 180,E1 -11451.755,E2 -11451.755} C_VEL
LIN {X 0,Y 399.425,Z 421.549,A -85,B 0,C 180,E1 -11452.773,E2 -11452.773} C_VEL
LIN {X 0,Y 400.751,Z 406.621,A -85,B 0,C 180,E1 -11453.787,E2 -11453.787} C_VEL
LIN {X 0,Y 401.234,Z 399.085,A -85,B 0,C 180,E1 -11454.212,E2 -11454.212} C_VEL
LIN {X 0,Y 397.885,Z 386.608,A -85,B 0,C 180,E1 -11455.065,E2 -11455.065} C_VEL
LIN {X 0,Y 393.203,Z 372.91,A -85,B 0,C 180,E1 -11455.905,E2 -11455.905} C_VEL
LIN {X 0,Y 389.424,Z 363.196,A -85,B 0,C 180,E1 -11456.437,E2 -11456.437} C_VEL
LIN {X 0,Y 389.282,Z 362.453,A -85,B 0,C 180,E1 -11456.472,E2 -11456.472} C_VEL
LIN {X 0,Y 389.43,Z 359.37,A -85,B 0,C 180,E1 -11459.974,E2 -11459.974} C_VEL
LIN {X 0,Y 389.507,Z 357.058,A -85,B 0,C 180,E1 -11462.772,E2 -11462.772} C_VEL
LIN {X 0,Y 389.626,Z 354.048,A -85,B 0,C 180,E1 -11466.53,E2 -11466.53} C_VEL
LIN {X 0,Y 389.655,Z 353.066,A -85,B 0,C 180,E1 -11467.824,E2 -11467.824} C_VEL
LIN {X 0,Y 389.769,Z 352.561,A -85,B 0,C 180,E1 -11469.164,E2 -11469.164} C_VEL
LIN {X 0,Y 390.008,Z 352.525,A -85,B 0,C 180,E1 -11472.368,E2 -11472.368} C_VEL
LIN {X 0,Y 390.044,Z 352.524,A -85,B 0,C 180,E1 -11475.354,E2 -11475.354} C_VEL
LIN {X 0,Y 390.03,Z 352.527,A -85,B 0,C 180,E1 -11478.186,E2 -11478.186} C_VEL
LIN {X 0,Y 390.091,Z 352.519,A -85,B 0,C 180,E1 -11480.908,E2 -11480.908} C_VEL
LIN {X 0,Y 390.084,Z 352.52,A -85,B 0,C 180,E1 -11484.793,E2 -11484.793} C_VEL
LIN {X 0,Y 390.032,Z 352.518,A -85,B 0,C 180,E1 -11487.874,E2 -11487.874} C_VEL
LIN {X 0,Y 390.064,Z 352.522,A -85,B 0,C 180,E1 -11490.891,E2 -11490.891} C_VEL
LIN {X 0,Y 390.11,Z 352.51,A -85,B 0,C 180,E1 -11494.382,E2 -11494.382} C_VEL
LIN {X 0,Y 390.038,Z 352.519,A -85,B 0,C 180,E1 -11497.766,E2 -11497.766} C_VEL
LIN {X 0,Y 390.104,Z 352.511,A -85,B 0,C 180,E1 -11501.078,E2 -11501.078} C_VEL
LIN {X 0,Y 390.138,Z 352.51,A -85,B 0,C 180,E1 -11504.323,E2 -11504.323} C_VEL
LIN {X 0,Y 390.176,Z 352.491,A -85,B 0,C 180,E1 -11507.517,E2 -11507.517} C_VEL
LIN {X 0,Y 390.313,Z 352.489,A -85,B 0,C 180,E1 -11511.718,E2 -11511.718} C_VEL
LIN {X 0,Y 390.328,Z 352.49,A -85,B 0,C 180,E1 -11513.798,E2 -11513.798} C_VEL
LIN {X 0,Y 390.419,Z 352.478,A -85,B 0,C 180,E1 -11517.937,E2 -11517.937} C_VEL
LIN {X 0,Y 390.548,Z 352.464,A -85,B 0,C 180,E1 -11520,E2 -11520} C_VEL
LIN {X 0,Y 390.314,Z 352.493,A -85,B 0,C 180,E1 -11523.096,E2 -11523.096} C_VEL
LIN {X 0,Y 390.328,Z 352.492,A -85,B 0,C 180,E1 -11526.202,E2 -11526.202} C_VEL
LIN {X 0,Y 390.312,Z 352.491,A -85,B 0,C 180,E1 -11528.282,E2 -11528.282} C_VEL
LIN {X 0,Y 390.169,Z 352.507,A -85,B 0,C 180,E1 -11532.483,E2 -11532.483} C_VEL
LIN {X 0,Y 390.137,Z 352.511,A -85,B 0,C 180,E1 -11535.677,E2 -11535.677} C_VEL
LIN {X 0,Y 390.103,Z 352.518,A -85,B 0,C 180,E1 -11538.922,E2 -11538.922} C_VEL
LIN {X 0,Y 390.037,Z 352.525,A -85,B 0,C 180,E1 -11542.234,E2 -11542.234} C_VEL
LIN {X 0,Y 390.117,Z 352.518,A -85,B 0,C 180,E1 -11545.744,E2 -11545.744} C_VEL
LIN {X 0,Y 390.063,Z 352.526,A -85,B 0,C 180,E1 -11549.109,E2 -11549.109} C_VEL
LIN {X 0,Y 390.042,Z 352.527,A -85,B 0,C 180,E1 -11552.721,E2 -11552.721} C_VEL
LIN {X 0,Y 390.055,Z 352.526,A -85,B 0,C 180,E1 -11555.826,E2 -11555.826} C_VEL
LIN {X 0,Y 390.062,Z 352.529,A -85,B 0,C 180,E1 -11558.105,E2 -11558.105} C_VEL
LIN {X 0,Y 390.696,Z 356.175,A -85,B 0,C 180,E1 -11560.931,E2 -11560.931} C_VEL
LIN {X 0,Y 391.523,Z 361.088,A -85,B 0,C 180,E1 -11564.432,E2 -11564.432} C_VEL
LIN {X 0,Y 392.127,Z 365.431,A -85,B 0,C 180,E1 -11567.293,E2 -11567.293} C_VEL
LIN {X 0,Y 392.201,Z 367.897,A -85,B 0,C 180,E1 -11568.817,E2 -11568.817} C_VEL
LIN {X 0,Y 391.607,Z 374.049,A -85,B 0,C 180,E1 -11572.398,E2 -11572.398} C_VEL
LIN {X 0,Y 391.142,Z 380.053,A -85,B 0,C 180,E1 -11575.743,E2 -11575.743} C_VEL
LIN {X 0,Y 390.597,Z 386.357,A -85,B 0,C 180,E1 -11579.15,E2 -11579.15} C_VEL
LIN {X 0,Y 390.047,Z 392.927,A -85,B 0,C 180,E1 -11582.648,E2 -11582.648} C_VEL
LIN {X 0,Y 389.98,Z 394.73,A -85,B 0,C 180,E1 -11583.592,E2 -11583.592} C_VEL
LIN {X 0,Y 391.363,Z 400.004,A -85,B 0,C 180,E1 -11583.809,E2 -11583.809} C_VEL
LIN {X 0,Y 395.447,Z 415.251,A -85,B 0,C 180,E1 -11584.551,E2 -11584.551} C_VEL
LIN {X 0,Y 398.526,Z 430.33,A -85,B 0,C 180,E1 -11585.42,E2 -11585.42} C_VEL
LIN {X 0,Y 399.911,Z 439.834,A -85,B 0,C 180,E1 -11586.042,E2 -11586.042} C_VEL
LIN {X 0,Y 398.675,Z 454.122,A -85,B 0,C 180,E1 -11586.955,E2 -11586.955} C_VEL
LIN {X 0,Y 397.108,Z 467.82,A -85,B 0,C 180,E1 -11588.046,E2 -11588.046} C_VEL
LIN {X 0,Y 395.557,Z 480.802,A -85,B 0,C 180,E1 -11589.322,E2 -11589.322} C_VEL
LIN {X 0,Y 394.113,Z 492.704,A -85,B 0,C 180,E1 -11590.738,E2 -11590.738} C_VEL
LIN {X 0,Y 392.79,Z 503.614,A -85,B 0,C 180,E1 -11592.292,E2 -11592.292} C_VEL
LIN {X 0,Y 391.564,Z 512.875,A -85,B 0,C 180,E1 -11593.848,E2 -11593.848} C_VEL
LIN {X 0,Y 390.54,Z 521.975,A -85,B 0,C 180,E1 -11595.674,E2 -11595.674} C_VEL
LIN {X 0,Y 389.837,Z 529.534,A -85,B 0,C 180,E1 -11597.507,E2 -11597.507} C_VEL
LIN {X 0,Y 389.179,Z 536.589,A -85,B 0,C 180,E1 -11599.597,E2 -11599.597} C_VEL
LIN {X 0,Y 388.914,Z 542.151,A -85,B 0,C 180,E1 -11601.688,E2 -11601.688} C_VEL
LIN {X 0,Y 388.773,Z 546.5,A -85,B 0,C 180,E1 -11603.855,E2 -11603.855} C_VEL
LIN {X 0,Y 388.695,Z 549.308,A -85,B 0,C 180,E1 -11605.853,E2 -11605.853} C_VEL
LIN {X 0,Y 388.779,Z 551.074,A -85,B 0,C 180,E1 -11607.929,E2 -11607.929} C_VEL
LIN {X 0,Y 388.743,Z 551.675,A -85,B 0,C 180,E1 -11610,E2 -11610} C_VEL
LIN {X 0,Y 388.78,Z 551.069,A -85,B 0,C 180,E1 -11612.072,E2 -11612.072} C_VEL
LIN {X 0,Y 388.7,Z 549.297,A -85,B 0,C 180,E1 -11614.148,E2 -11614.148} C_VEL
LIN {X 0,Y 388.833,Z 546.348,A -85,B 0,C 180,E1 -11616.226,E2 -11616.226} C_VEL
LIN {X 0,Y 388.914,Z 542.139,A -85,B 0,C 180,E1 -11618.313,E2 -11618.313} C_VEL
LIN {X 0,Y 389.18,Z 536.57,A -85,B 0,C 180,E1 -11620.404,E2 -11620.404} C_VEL
LIN {X 0,Y 389.844,Z 529.502,A -85,B 0,C 180,E1 -11622.494,E2 -11622.494} C_VEL
LIN {X 0,Y 390.542,Z 521.94,A -85,B 0,C 180,E1 -11624.326,E2 -11624.326} C_VEL
LIN {X 0,Y 391.571,Z 512.839,A -85,B 0,C 180,E1 -11626.153,E2 -11626.153} C_VEL
LIN {X 0,Y 392.985,Z 501.919,A -85,B 0,C 180,E1 -11627.969,E2 -11627.969} C_VEL
LIN {X 0,Y 394.426,Z 489.754,A -85,B 0,C 180,E1 -11629.64,E2 -11629.64} C_VEL
LIN {X 0,Y 395.973,Z 477.147,A -85,B 0,C 180,E1 -11631.064,E2 -11631.064} C_VEL
LIN {X 0,Y 397.625,Z 463.333,A -85,B 0,C 180,E1 -11632.335,E2 -11632.335} C_VEL
LIN {X 0,Y 399.11,Z 449.577,A -85,B 0,C 180,E1 -11633.355,E2 -11633.355} C_VEL
LIN {X 0,Y 399.922,Z 439.638,A -85,B 0,C 180,E1 -11633.962,E2 -11633.962} C_VEL
LIN {X 0,Y 397.483,Z 424.636,A -85,B 0,C 180,E1 -11634.915,E2 -11634.915} C_VEL
LIN {X 0,Y 393.956,Z 409.409,A -85,B 0,C 180,E1 -11635.742,E2 -11635.742} C_VEL
LIN {X 0,Y 389.962,Z 394.694,A -85,B 0,C 180,E1 -11636.405,E2 -11636.405} C_VEL
LIN {X 0,Y 390.502,Z 387.428,A -85,B 0,C 180,E1 -11640.261,E2 -11640.261} C_VEL
LIN {X 0,Y 391.04,Z 380.731,A -85,B 0,C 180,E1 -11643.859,E2 -11643.859} C_VEL
LIN {X 0,Y 391.52,Z 375.116,A -85,B 0,C 180,E1 -11646.967,E2 -11646.967} C_VEL
LIN {X 0,Y 392.052,Z 369.461,A -85,B 0,C 180,E1 -11650.192,E2 -11650.192} C_VEL
LIN {X 0,Y 392.191,Z 367.225,A -85,B 0,C 180,E1 -11651.532,E2 -11651.532} C_VEL
LIN {X 0,Y 391.861,Z 363.089,A -85,B 0,C 180,E1 -11654.16,E2 -11654.16} C_VEL
LIN {X 0,Y 391.067,Z 358.333,A -85,B 0,C 180,E1 -11657.462,E2 -11657.462} C_VEL
LIN {X 0,Y 390.298,Z 353.695,A -85,B 0,C 180,E1 -11660.933,E2 -11660.933} C_VEL
LIN {X 0,Y 390.066,Z 352.526,A -85,B 0,C 180,E1 -11661.896,E2 -11661.896} C_VEL
LIN {X 0,Y 390.088,Z 352.524,A -85,B 0,C 180,E1 -11664.794,E2 -11664.794} C_VEL
LIN {X 0,Y 390.026,Z 352.528,A -85,B 0,C 180,E1 -11668.496,E2 -11668.496} C_VEL
LIN {X 0,Y 390.12,Z 352.517,A -85,B 0,C 180,E1 -11672.07,E2 -11672.07} C_VEL
LIN {X 0,Y 390.083,Z 352.523,A -85,B 0,C 180,E1 -11675.52,E2 -11675.52} C_VEL
LIN {X 0,Y 390.058,Z 352.524,A -85,B 0,C 180,E1 -11678.878,E2 -11678.878} C_VEL
LIN {X 0,Y 390.131,Z 352.514,A -85,B 0,C 180,E1 -11682.167,E2 -11682.167} C_VEL
LIN {X 0,Y 390.147,Z 352.514,A -85,B 0,C 180,E1 -11685.393,E2 -11685.393} C_VEL
LIN {X 0,Y 390.151,Z 352.514,A -85,B 0,C 180,E1 -11688.571,E2 -11688.571} C_VEL
LIN {X 0,Y 390.347,Z 352.49,A -85,B 0,C 180,E1 -11691.993,E2 -11691.993} C_VEL
LIN {X 0,Y 390.23,Z 352.502,A -85,B 0,C 180,E1 -11694.834,E2 -11694.834} C_VEL
LIN {X 0,Y 390.424,Z 352.477,A -85,B 0,C 180,E1 -11697.937,E2 -11697.937} C_VEL
LIN {X 0,Y 390.552,Z 352.46,A -85,B 0,C 180,E1 -11700,E2 -11700} C_VEL
LIN {X 0,Y 390.318,Z 352.488,A -85,B 0,C 180,E1 -11703.097,E2 -11703.097} C_VEL
LIN {X 0,Y 390.314,Z 352.486,A -85,B 0,C 180,E1 -11706.628,E2 -11706.628} C_VEL
LIN {X 0,Y 390.209,Z 352.504,A -85,B 0,C 180,E1 -11709.329,E2 -11709.329} C_VEL
LIN {X 0,Y 390.174,Z 352.485,A -85,B 0,C 180,E1 -11712.483,E2 -11712.483} C_VEL
LIN {X 0,Y 390.143,Z 352.51,A -85,B 0,C 180,E1 -11715.677,E2 -11715.677} C_VEL
LIN {X 0,Y 390.109,Z 352.509,A -85,B 0,C 180,E1 -11718.922,E2 -11718.922} C_VEL
LIN {X 0,Y 390.04,Z 352.518,A -85,B 0,C 180,E1 -11722.234,E2 -11722.234} C_VEL
LIN {X 0,Y 390.122,Z 352.508,A -85,B 0,C 180,E1 -11725.743,E2 -11725.743} C_VEL
LIN {X 0,Y 390.062,Z 352.52,A -85,B 0,C 180,E1 -11729.109,E2 -11729.109} C_VEL
LIN {X 0,Y 390.046,Z 352.516,A -85,B 0,C 180,E1 -11732.721,E2 -11732.721} C_VEL
LIN {X 0,Y 390.06,Z 352.522,A -85,B 0,C 180,E1 -11735.825,E2 -11735.825} C_VEL
LIN {X 0,Y 390.075,Z 352.522,A -85,B 0,C 180,E1 -11739.219,E2 -11739.219} C_VEL
LIN {X 0,Y 390.046,Z 352.528,A -85,B 0,C 180,E1 -11742.374,E2 -11742.374} C_VEL
LIN {X 0,Y 390.047,Z 352.529,A -85,B 0,C 180,E1 -11745.354,E2 -11745.354} C_VEL
LIN {X 0,Y 389.978,Z 352.538,A -85,B 0,C 180,E1 -11748.179,E2 -11748.179} C_VEL
LIN {X 0,Y 389.76,Z 352.563,A -85,B 0,C 180,E1 -11750.868,E2 -11750.868} C_VEL
LIN {X 0,Y 389.651,Z 353.251,A -85,B 0,C 180,E1 -11752.525,E2 -11752.525} C_VEL
LIN {X 0,Y 389.551,Z 355.946,A -85,B 0,C 180,E1 -11755.994,E2 -11755.994} C_VEL
LIN {X 0,Y 389.502,Z 357.957,A -85,B 0,C 180,E1 -11758.448,E2 -11758.448} C_VEL
LIN {X 0,Y 389.403,Z 359.959,A -85,B 0,C 180,E1 -11760.836,E2 -11760.836} C_VEL
LIN {X 0,Y 389.327,Z 362.608,A -85,B 0,C 180,E1 -11763.643,E2 -11763.643} C_VEL
LIN {X 0,Y 391.429,Z 368.376,A -85,B 0,C 180,E1 -11763.935,E2 -11763.935} C_VEL
LIN {X 0,Y 396.201,Z 381.415,A -85,B 0,C 180,E1 -11764.704,E2 -11764.704} C_VEL
LIN {X 0,Y 400.544,Z 396.026,A -85,B 0,C 180,E1 -11765.676,E2 -11765.676} C_VEL
LIN {X 0,Y 401.203,Z 398.469,A -85,B 0,C 180,E1 -11765.851,E2 -11765.851} C_VEL
LIN {X 0,Y 400.155,Z 413.43,A -85,B 0,C 180,E1 -11766.743,E2 -11766.743} C_VEL
LIN {X 0,Y 398.881,Z 426.693,A -85,B 0,C 180,E1 -11767.739,E2 -11767.739} C_VEL
LIN {X 0,Y 397.465,Z 439.146,A -85,B 0,C 180,E1 -11768.883,E2 -11768.883} C_VEL
LIN {X 0,Y 395.939,Z 451.748,A -85,B 0,C 180,E1 -11770.29,E2 -11770.29} C_VEL
LIN {X 0,Y 394.49,Z 463.165,A -85,B 0,C 180,E1 -11771.834,E2 -11771.834} C_VEL
LIN {X 0,Y 393.207,Z 472.766,A -85,B 0,C 180,E1 -11773.382,E2 -11773.382} C_VEL
LIN {X 0,Y 391.976,Z 482.168,A -85,B 0,C 180,E1 -11775.197,E2 -11775.197} C_VEL
LIN {X 0,Y 391.124,Z 489.981,A -85,B 0,C 180,E1 -11777.02,E2 -11777.02} C_VEL
LIN {X 0,Y 390.146,Z 497.281,A -85,B 0,C 180,E1 -11779.097,E2 -11779.097} C_VEL
LIN {X 0,Y 389.59,Z 503.061,A -85,B 0,C 180,E1 -11781.179,E2 -11781.179} C_VEL
LIN {X 0,Y 389.157,Z 507.65,A -85,B 0,C 180,E1 -11783.353,E2 -11783.353} C_VEL
LIN {X 0,Y 388.973,Z 509.949,A -85,B 0,C 180,E1 -11784.816,E2 -11784.816} C_VEL
LIN {X 0,Y 388.931,Z 512.234,A -85,B 0,C 180,E1 -11786.892,E2 -11786.892} C_VEL
LIN {X 0,Y 388.783,Z 513.408,A -85,B 0,C 180,E1 -11788.964,E2 -11788.964} C_VEL
LIN {X 0,Y 388.783,Z 513.423,A -85,B 0,C 180,E1 -11791.035,E2 -11791.035} C_VEL
LIN {X 0,Y 388.93,Z 512.311,A -85,B 0,C 180,E1 -11793.107,E2 -11793.107} C_VEL
LIN {X 0,Y 388.971,Z 510.086,A -85,B 0,C 180,E1 -11795.183,E2 -11795.183} C_VEL
LIN {X 0,Y 389.24,Z 506.678,A -85,B 0,C 180,E1 -11797.261,E2 -11797.261} C_VEL
LIN {X 0,Y 389.705,Z 502.007,A -85,B 0,C 180,E1 -11799.34,E2 -11799.34} C_VEL
LIN {X 0,Y 390.274,Z 495.956,A -85,B 0,C 180,E1 -11801.425,E2 -11801.425} C_VEL
LIN {X 0,Y 391.266,Z 488.32,A -85,B 0,C 180,E1 -11803.503,E2 -11803.503} C_VEL
LIN {X 0,Y 392.214,Z 480.18,A -85,B 0,C 180,E1 -11805.325,E2 -11805.325} C_VEL
LIN {X 0,Y 393.574,Z 470.358,A -85,B 0,C 180,E1 -11807.135,E2 -11807.135} C_VEL
LIN {X 0,Y 394.82,Z 460.285,A -85,B 0,C 180,E1 -11808.687,E2 -11808.687} C_VEL
LIN {X 0,Y 395.099,Z 458.325,A -85,B 0,C 180,E1 -11808.957,E2 -11808.957} C_VEL
LIN {X 0,Y 395.032,Z 454.091,A -85,B 0,C 180,E1 -11809.555,E2 -11809.555} C_VEL
LIN {X 0,Y 391.769,Z 441.465,A -85,B 0,C 180,E1 -11811.332,E2 -11811.332} C_VEL
LIN {X 0,Y 391.359,Z 436.817,A -85,B 0,C 180,E1 -11811.86,E2 -11811.86} C_VEL
LIN {X 0,Y 391.46,Z 435.181,A -85,B 0,C 180,E1 -11812.019,E2 -11812.019} C_VEL
LIN {X 0,Y 392.908,Z 421.89,A -85,B 0,C 180,E1 -11813.173,E2 -11813.173} C_VEL
LIN {X 0,Y 394.255,Z 406.961,A -85,B 0,C 180,E1 -11814.204,E2 -11814.204} C_VEL
LIN {X 0,Y 394.652,Z 400.063,A -85,B 0,C 180,E1 -11814.607,E2 -11814.607} C_VEL
LIN {X 0,Y 390.599,Z 385.804,A -85,B 0,C 180,E1 -11815.622,E2 -11815.622} C_VEL
LIN {X 0,Y 385.793,Z 372.079,A -85,B 0,C 180,E1 -11816.48,E2 -11816.48} C_VEL
LIN {X 0,Y 382.374,Z 363.53,A -85,B 0,C 180,E1 -11816.964,E2 -11816.964} C_VEL
LIN {X 0,Y 382.264,Z 362.788,A -85,B 0,C 180,E1 -11817.026,E2 -11817.026} C_VEL
LIN {X 0,Y 382.417,Z 359.394,A -85,B 0,C 180,E1 -11820.969,E2 -11820.969} C_VEL
LIN {X 0,Y 382.512,Z 356.761,A -85,B 0,C 180,E1 -11824.229,E2 -11824.229} C_VEL
LIN {X 0,Y 382.618,Z 353.977,A -85,B 0,C 180,E1 -11827.83,E2 -11827.83} C_VEL
LIN {X 0,Y 382.65,Z 353.449,A -85,B 0,C 180,E1 -11828.642,E2 -11828.642} C_VEL
LIN {X 0,Y 382.891,Z 353.413,A -85,B 0,C 180,E1 -11831.359,E2 -11831.359} C_VEL
LIN {X 0,Y 382.993,Z 353.402,A -85,B 0,C 180,E1 -11834.303,E2 -11834.303} C_VEL
LIN {X 0,Y 383.008,Z 353.402,A -85,B 0,C 180,E1 -11837.24,E2 -11837.24} C_VEL
LIN {X 0,Y 383.015,Z 353.402,A -85,B 0,C 180,E1 -11840.413,E2 -11840.413} C_VEL
LIN {X 0,Y 383.025,Z 353.4,A -85,B 0,C 180,E1 -11844.044,E2 -11844.044} C_VEL
LIN {X 0,Y 382.987,Z 353.394,A -85,B 0,C 180,E1 -11847.577,E2 -11847.577} C_VEL
LIN {X 0,Y 382.997,Z 353.402,A -85,B 0,C 180,E1 -11850.3,E2 -11850.3} C_VEL
LIN {X 0,Y 383.055,Z 353.381,A -85,B 0,C 180,E1 -11852.698,E2 -11852.698} C_VEL
LIN {X 0,Y 383.05,Z 353.393,A -85,B 0,C 180,E1 -11855.039,E2 -11855.039} C_VEL
LIN {X 0,Y 382.991,Z 353.392,A -85,B 0,C 180,E1 -11858.469,E2 -11858.469} C_VEL
LIN {X 0,Y 383.061,Z 353.391,A -85,B 0,C 180,E1 -11861.826,E2 -11861.826} C_VEL
LIN {X 0,Y 383.11,Z 353.38,A -85,B 0,C 180,E1 -11865.118,E2 -11865.118} C_VEL
LIN {X 0,Y 383.106,Z 353.379,A -85,B 0,C 180,E1 -11868.358,E2 -11868.358} C_VEL
LIN {X 0,Y 383.302,Z 353.362,A -85,B 0,C 180,E1 -11871.932,E2 -11871.932} C_VEL
LIN {X 0,Y 383.198,Z 353.377,A -85,B 0,C 180,E1 -11874.738,E2 -11874.738} C_VEL
LIN {X 0,Y 383.386,Z 353.354,A -85,B 0,C 180,E1 -11877.899,E2 -11877.899} C_VEL
LIN {X 0,Y 383.517,Z 353.34,A -85,B 0,C 180,E1 -11880,E2 -11880} C_VEL
LIN {X 0,Y 383.251,Z 353.373,A -85,B 0,C 180,E1 -11883.154,E2 -11883.154} C_VEL
LIN {X 0,Y 383.285,Z 353.369,A -85,B 0,C 180,E1 -11886.316,E2 -11886.316} C_VEL
LIN {X 0,Y 383.258,Z 353.37,A -85,B 0,C 180,E1 -11888.436,E2 -11888.436} C_VEL
LIN {X 0,Y 383.096,Z 353.389,A -85,B 0,C 180,E1 -11891.642,E2 -11891.642} C_VEL
LIN {X 0,Y 383.108,Z 353.387,A -85,B 0,C 180,E1 -11894.882,E2 -11894.882} C_VEL
LIN {X 0,Y 383.087,Z 353.39,A -85,B 0,C 180,E1 -11898.172,E2 -11898.172} C_VEL
LIN {X 0,Y 382.991,Z 353.405,A -85,B 0,C 180,E1 -11901.531,E2 -11901.531} C_VEL
LIN {X 0,Y 383.05,Z 353.398,A -85,B 0,C 180,E1 -11904.96,E2 -11904.96} C_VEL
LIN {X 0,Y 383.047,Z 353.398,A -85,B 0,C 180,E1 -11908.492,E2 -11908.492} C_VEL
LIN {X 0,Y 383.011,Z 353.401,A -85,B 0,C 180,E1 -11912.149,E2 -11912.149} C_VEL
LIN {X 0,Y 383.016,Z 353.403,A -85,B 0,C 180,E1 -11914.668,E2 -11914.668} C_VEL
LIN {X 0,Y 383.025,Z 353.497,A -85,B 0,C 180,E1 -11917.704,E2 -11917.704} C_VEL
LIN {X 0,Y 383.836,Z 358.145,A -85,B 0,C 180,E1 -11921.349,E2 -11921.349} C_VEL
LIN {X 0,Y 384.578,Z 362.592,A -85,B 0,C 180,E1 -11924.545,E2 -11924.545} C_VEL
LIN {X 0,Y 385.069,Z 366.064,A -85,B 0,C 180,E1 -11926.89,E2 -11926.89} C_VEL
LIN {X 0,Y 385.175,Z 369.295,A -85,B 0,C 180,E1 -11928.939,E2 -11928.939} C_VEL
LIN {X 0,Y 384.685,Z 374.061,A -85,B 0,C 180,E1 -11931.775,E2 -11931.775} C_VEL
LIN {X 0,Y 384.144,Z 380.472,A -85,B 0,C 180,E1 -11935.449,E2 -11935.449} C_VEL
LIN {X 0,Y 383.545,Z 387.131,A -85,B 0,C 180,E1 -11939.132,E2 -11939.132} C_VEL
LIN {X 0,Y 382.948,Z 394.32,A -85,B 0,C 180,E1 -11943.062,E2 -11943.062} C_VEL
LIN {X 0,Y 384.495,Z 400.062,A -85,B 0,C 180,E1 -11943.314,E2 -11943.314} C_VEL
LIN {X 0,Y 388.556,Z 415.12,A -85,B 0,C 180,E1 -11944.076,E2 -11944.076} C_VEL
LIN {X 0,Y 391.665,Z 430.009,A -85,B 0,C 180,E1 -11944.963,E2 -11944.963} C_VEL
LIN {X 0,Y 393.27,Z 441.434,A -85,B 0,C 180,E1 -11945.731,E2 -11945.731} C_VEL
LIN {X 0,Y 391.954,Z 455.367,A -85,B 0,C 180,E1 -11946.662,E2 -11946.662} C_VEL
LIN {X 0,Y 390.303,Z 468.906,A -85,B 0,C 180,E1 -11947.782,E2 -11947.782} C_VEL
LIN {X 0,Y 388.711,Z 481.635,A -85,B 0,C 180,E1 -11949.079,E2 -11949.079} C_VEL
LIN {X 0,Y 387.204,Z 493.437,A -85,B 0,C 180,E1 -11950.532,E2 -11950.532} C_VEL
LIN {X 0,Y 385.715,Z 504.907,A -85,B 0,C 180,E1 -11952.23,E2 -11952.23} C_VEL
LIN {X 0,Y 384.491,Z 513.895,A -85,B 0,C 180,E1 -11953.815,E2 -11953.815} C_VEL
LIN {X 0,Y 383.456,Z 522.758,A -85,B 0,C 180,E1 -11955.675,E2 -11955.675} C_VEL
LIN {X 0,Y 382.827,Z 529.183,A -85,B 0,C 180,E1 -11957.274,E2 -11957.274} C_VEL
LIN {X 0,Y 382.138,Z 536.24,A -85,B 0,C 180,E1 -11959.403,E2 -11959.403} C_VEL
LIN {X 0,Y 381.824,Z 541.8,A -85,B 0,C 180,E1 -11961.533,E2 -11961.533} C_VEL
LIN {X 0,Y 381.672,Z 546.427,A -85,B 0,C 180,E1 -11963.901,E2 -11963.901} C_VEL
LIN {X 0,Y 381.619,Z 548.961,A -85,B 0,C 180,E1 -11965.776,E2 -11965.776} C_VEL
LIN {X 0,Y 381.678,Z 550.726,A -85,B 0,C 180,E1 -11967.89,E2 -11967.89} C_VEL
LIN {X 0,Y 381.673,Z 551.328,A -85,B 0,C 180,E1 -11970,E2 -11970} C_VEL
LIN {X 0,Y 381.679,Z 550.72,A -85,B 0,C 180,E1 -11972.111,E2 -11972.111} C_VEL
LIN {X 0,Y 381.626,Z 548.949,A -85,B 0,C 180,E1 -11974.225,E2 -11974.225} C_VEL
LIN {X 0,Y 381.737,Z 545.998,A -85,B 0,C 180,E1 -11976.342,E2 -11976.342} C_VEL
LIN {X 0,Y 381.824,Z 541.787,A -85,B 0,C 180,E1 -11978.468,E2 -11978.468} C_VEL
LIN {X 0,Y 382.139,Z 536.218,A -85,B 0,C 180,E1 -11980.598,E2 -11980.598} C_VEL
LIN {X 0,Y 382.832,Z 529.148,A -85,B 0,C 180,E1 -11982.727,E2 -11982.727} C_VEL
LIN {X 0,Y 383.723,Z 520.356,A -85,B 0,C 180,E1 -11984.858,E2 -11984.858} C_VEL
LIN {X 0,Y 384.818,Z 511.029,A -85,B 0,C 180,E1 -11986.717,E2 -11986.717} C_VEL
LIN {X 0,Y 386.147,Z 501.613,A -85,B 0,C 180,E1 -11988.29,E2 -11988.29} C_VEL
LIN {X 0,Y 387.515,Z 490.518,A -85,B 0,C 180,E1 -11989.853,E2 -11989.853} C_VEL
LIN {X 0,Y 389.132,Z 478.02,A -85,B 0,C 180,E1 -11991.314,E2 -11991.314} C_VEL
LIN {X 0,Y 390.839,Z 464.508,A -85,B 0,C 180,E1 -11992.605,E2 -11992.605} C_VEL
LIN {X 0,Y 392.501,Z 449.939,A -85,B 0,C 180,E1 -11993.721,E2 -11993.721} C_VEL
LIN {X 0,Y 393.276,Z 440.743,A -85,B 0,C 180,E1 -11994.302,E2 -11994.302} C_VEL
LIN {X 0,Y 391.361,Z 428.255,A -85,B 0,C 180,E1 -11995.144,E2 -11995.144} C_VEL
LIN {X 0,Y 388.153,Z 413.513,A -85,B 0,C 180,E1 -11996.005,E2 -11996.005} C_VEL
LIN {X 0,Y 383.915,Z 397.806,A -85,B 0,C 180,E1 -11996.772,E2 -11996.772} C_VEL
LIN {X 0,Y 382.96,Z 394.33,A -85,B 0,C 180,E1 -11996.936,E2 -11996.936} C_VEL
LIN {X 0,Y 383.476,Z 387.723,A -85,B 0,C 180,E1 -12000.529,E2 -12000.529} C_VEL
LIN {X 0,Y 384.018,Z 381.533,A -85,B 0,C 180,E1 -12003.931,E2 -12003.931} C_VEL
LIN {X 0,Y 384.527,Z 375.961,A -85,B 0,C 180,E1 -12007.096,E2 -12007.096} C_VEL
LIN {X 0,Y 385.149,Z 369.179,A -85,B 0,C 180,E1 -12011.065,E2 -12011.065} C_VEL
LIN {X 0,Y 385.056,Z 365.951,A -85,B 0,C 180,E1 -12013.107,E2 -12013.107} C_VEL
LIN {X 0,Y 384.447,Z 361.723,A -85,B 0,C 180,E1 -12015.999,E2 -12015.999} C_VEL
LIN {X 0,Y 383.789,Z 357.955,A -85,B 0,C 180,E1 -12018.758,E2 -12018.758} C_VEL
LIN {X 0,Y 383.056,Z 353.726,A -85,B 0,C 180,E1 -12022.086,E2 -12022.086} C_VEL
LIN {X 0,Y 382.999,Z 353.407,A -85,B 0,C 180,E1 -12022.732,E2 -12022.732} C_VEL
LIN {X 0,Y 383.02,Z 353.403,A -85,B 0,C 180,E1 -12025.66,E2 -12025.66} C_VEL
LIN {X 0,Y 382.985,Z 353.404,A -85,B 0,C 180,E1 -12029.082,E2 -12029.082} C_VEL
LIN {X 0,Y 383.059,Z 353.396,A -85,B 0,C 180,E1 -12032.698,E2 -12032.698} C_VEL
LIN {X 0,Y 383.036,Z 353.398,A -85,B 0,C 180,E1 -12036.193,E2 -12036.193} C_VEL
LIN {X 0,Y 383.058,Z 353.396,A -85,B 0,C 180,E1 -12039.599,E2 -12039.599} C_VEL
LIN {X 0,Y 383.108,Z 353.392,A -85,B 0,C 180,E1 -12042.932,E2 -12042.932} C_VEL
LIN {X 0,Y 383.128,Z 353.39,A -85,B 0,C 180,E1 -12046.464,E2 -12046.464} C_VEL
LIN {X 0,Y 383.155,Z 353.387,A -85,B 0,C 180,E1 -12050.498,E2 -12050.498} C_VEL
LIN {X 0,Y 383.277,Z 353.369,A -85,B 0,C 180,E1 -12052.625,E2 -12052.625} C_VEL
LIN {X 0,Y 383.202,Z 353.377,A -85,B 0,C 180,E1 -12054.739,E2 -12054.739} C_VEL
LIN {X 0,Y 383.391,Z 353.353,A -85,B 0,C 180,E1 -12057.899,E2 -12057.899} C_VEL
LIN {X 0,Y 383.521,Z 353.336,A -85,B 0,C 180,E1 -12060,E2 -12060} C_VEL
LIN {X 0,Y 383.254,Z 353.368,A -85,B 0,C 180,E1 -12063.154,E2 -12063.154} C_VEL
LIN {X 0,Y 383.274,Z 353.363,A -85,B 0,C 180,E1 -12066.622,E2 -12066.622} C_VEL
LIN {X 0,Y 383.264,Z 353.369,A -85,B 0,C 180,E1 -12068.436,E2 -12068.436} C_VEL
LIN {X 0,Y 383.101,Z 353.375,A -85,B 0,C 180,E1 -12071.642,E2 -12071.642} C_VEL
LIN {X 0,Y 383.114,Z 353.38,A -85,B 0,C 180,E1 -12074.882,E2 -12074.882} C_VEL
LIN {X 0,Y 383.066,Z 353.389,A -85,B 0,C 180,E1 -12078.174,E2 -12078.174} C_VEL
LIN {X 0,Y 382.995,Z 353.39,A -85,B 0,C 180,E1 -12081.531,E2 -12081.531} C_VEL
LIN {X 0,Y 383.054,Z 353.393,A -85,B 0,C 180,E1 -12084.96,E2 -12084.96} C_VEL
LIN {X 0,Y 383.033,Z 353.387,A -85,B 0,C 180,E1 -12088.27,E2 -12088.27} C_VEL
LIN {X 0,Y 383.012,Z 353.394,A -85,B 0,C 180,E1 -12092.15,E2 -12092.15} C_VEL
LIN {X 0,Y 383.021,Z 353.393,A -85,B 0,C 180,E1 -12094.668,E2 -12094.668} C_VEL
LIN {X 0,Y 383.005,Z 353.404,A -85,B 0,C 180,E1 -12097.904,E2 -12097.904} C_VEL
LIN {X 0,Y 382.987,Z 353.405,A -85,B 0,C 180,E1 -12101.347,E2 -12101.347} C_VEL
LIN {X 0,Y 382.999,Z 353.406,A -85,B 0,C 180,E1 -12104.303,E2 -12104.303} C_VEL
LIN {X 0,Y 382.977,Z 353.41,A -85,B 0,C 180,E1 -12107.235,E2 -12107.235} C_VEL
LIN {X 0,Y 382.747,Z 353.436,A -85,B 0,C 180,E1 -12110.462,E2 -12110.462} C_VEL
LIN {X 0,Y 382.652,Z 353.449,A -85,B 0,C 180,E1 -12111.357,E2 -12111.357} C_VEL
LIN {X 0,Y 382.574,Z 355.266,A -85,B 0,C 180,E1 -12113.995,E2 -12113.995} C_VEL
LIN {X 0,Y 382.477,Z 358.282,A -85,B 0,C 180,E1 -12117.8,E2 -12117.8} C_VEL
LIN {X 0,Y 382.396,Z 360.304,A -85,B 0,C 180,E1 -12120.249,E2 -12120.249} C_VEL
LIN {X 0,Y 382.316,Z 362.942,A -85,B 0,C 180,E1 -12123.119,E2 -12123.119} C_VEL
LIN {X 0,Y 383.281,Z 365.872,A -85,B 0,C 180,E1 -12123.265,E2 -12123.265} C_VEL
LIN {X 0,Y 388.966,Z 380.819,A -85,B 0,C 180,E1 -12124.159,E2 -12124.159} C_VEL
LIN {X 0,Y 393.364,Z 395.264,A -85,B 0,C 180,E1 -12125.139,E2 -12125.139} C_VEL
LIN {X 0,Y 394.749,Z 400.531,A -85,B 0,C 180,E1 -12125.527,E2 -12125.527} C_VEL
LIN {X 0,Y 393.626,Z 414.182,A -85,B 0,C 180,E1 -12126.362,E2 -12126.362} C_VEL
LIN {X 0,Y 392.16,Z 428.601,A -85,B 0,C 180,E1 -12127.476,E2 -12127.476} C_VEL
LIN {X 0,Y 390.558,Z 442.029,A -85,B 0,C 180,E1 -12128.768,E2 -12128.768} C_VEL
LIN {X 0,Y 389.11,Z 453.296,A -85,B 0,C 180,E1 -12130.085,E2 -12130.085} C_VEL
LIN {X 0,Y 387.74,Z 463.517,A -85,B 0,C 180,E1 -12131.506,E2 -12131.506} C_VEL
LIN {X 0,Y 386.387,Z 473.118,A -85,B 0,C 180,E1 -12133.08,E2 -12133.08} C_VEL
LIN {X 0,Y 385.101,Z 482.519,A -85,B 0,C 180,E1 -12134.926,E2 -12134.926} C_VEL
LIN {X 0,Y 384.185,Z 490.332,A -85,B 0,C 180,E1 -12136.781,E2 -12136.781} C_VEL
LIN {X 0,Y 383.161,Z 497.632,A -85,B 0,C 180,E1 -12138.895,E2 -12138.895} C_VEL
LIN {X 0,Y 382.561,Z 503.411,A -85,B 0,C 180,E1 -12141.016,E2 -12141.016} C_VEL
LIN {X 0,Y 382.202,Z 506.833,A -85,B 0,C 180,E1 -12142.604,E2 -12142.604} C_VEL
LIN {X 0,Y 381.919,Z 510.296,A -85,B 0,C 180,E1 -12144.72,E2 -12144.72} C_VEL
LIN {X 0,Y 381.836,Z 512.582,A -85,B 0,C 180,E1 -12146.834,E2 -12146.834} C_VEL
LIN {X 0,Y 381.714,Z 513.755,A -85,B 0,C 180,E1 -12148.945,E2 -12148.945} C_VEL
LIN {X 0,Y 381.715,Z 513.77,A -85,B 0,C 180,E1 -12151.055,E2 -12151.055} C_VEL
LIN {X 0,Y 381.835,Z 512.659,A -85,B 0,C 180,E1 -12153.165,E2 -12153.165} C_VEL
LIN {X 0,Y 381.918,Z 510.433,A -85,B 0,C 180,E1 -12155.279,E2 -12155.279} C_VEL
LIN {X 0,Y 382.197,Z 507.025,A -85,B 0,C 180,E1 -12157.395,E2 -12157.395} C_VEL
LIN {X 0,Y 382.669,Z 502.355,A -85,B 0,C 180,E1 -12159.514,E2 -12159.514} C_VEL
LIN {X 0,Y 383.295,Z 496.303,A -85,B 0,C 180,E1 -12161.636,E2 -12161.636} C_VEL
LIN {X 0,Y 384.208,Z 489.713,A -85,B 0,C 180,E1 -12163.487,E2 -12163.487} C_VEL
LIN {X 0,Y 385.348,Z 480.527,A -85,B 0,C 180,E1 -12165.605,E2 -12165.605} C_VEL
LIN {X 0,Y 386.773,Z 470.704,A -85,B 0,C 180,E1 -12167.446,E2 -12167.446} C_VEL
LIN {X 0,Y 388.314,Z 459.083,A -85,B 0,C 180,E1 -12169.242,E2 -12169.242} C_VEL
LIN {X 0,Y 389.894,Z 447.521,A -85,B 0,C 180,E1 -12170.716,E2 -12170.716} C_VEL
LIN {X 0,Y 391.46,Z 435.181,A -85,B 0,C 180,E1 -12172.019,E2 -12172.019} C_VEL
LIN {X 0,Y 391.395,Z 430.328,A -85,B 0,C 180,E1 -12172.507,E2 -12172.507} C_VEL
LIN {X 0,Y 389.614,Z 422.363,A -85,B 0,C 180,E1 -12173.354,E2 -12173.354} C_VEL
LIN {X 0,Y 387.724,Z 414.233,A -85,B 0,C 180,E1 -12174.141,E2 -12174.141} C_VEL
LIN {X 0,Y 387.63,Z 408.98,A -85,B 0,C 180,E1 -12174.528,E2 -12174.528} C_VEL
LIN {X 0,Y 388.19,Z 402.187,A -85,B 0,C 180,E1 -12174.932,E2 -12174.932} C_VEL
LIN {X 0,Y 384.45,Z 388.57,A -85,B 0,C 180,E1 -12175.944,E2 -12175.944} C_VEL
LIN {X 0,Y 379.959,Z 375.409,A -85,B 0,C 180,E1 -12176.82,E2 -12176.82} C_VEL
LIN {X 0,Y 375.382,Z 364.14,A -85,B 0,C 180,E1 -12177.502,E2 -12177.502} C_VEL
LIN {X 0,Y 375.219,Z 363.161,A -85,B 0,C 180,E1 -12177.567,E2 -12177.567} C_VEL
LIN {X 0,Y 375.341,Z 360.612,A -85,B 0,C 180,E1 -12180.535,E2 -12180.535} C_VEL
LIN {X 0,Y 375.446,Z 358.729,A -85,B 0,C 180,E1 -12182.877,E2 -12182.877} C_VEL
LIN {X 0,Y 375.534,Z 355.961,A -85,B 0,C 180,E1 -12186.416,E2 -12186.416} C_VEL
LIN {X 0,Y 375.602,Z 354.632,A -85,B 0,C 180,E1 -12188.198,E2 -12188.198} C_VEL
LIN {X 0,Y 375.796,Z 354.298,A -85,B 0,C 180,E1 -12190.885,E2 -12190.885} C_VEL
LIN {X 0,Y 375.917,Z 354.281,A -85,B 0,C 180,E1 -12193.767,E2 -12193.767} C_VEL
LIN {X 0,Y 375.932,Z 354.282,A -85,B 0,C 180,E1 -12196.81,E2 -12196.81} C_VEL
LIN {X 0,Y 375.963,Z 354.281,A -85,B 0,C 180,E1 -12200.537,E2 -12200.537} C_VEL
LIN {X 0,Y 375.963,Z 354.279,A -85,B 0,C 180,E1 -12203.495,E2 -12203.495} C_VEL
LIN {X 0,Y 375.961,Z 354.273,A -85,B 0,C 180,E1 -12205.888,E2 -12205.888} C_VEL
LIN {X 0,Y 375.967,Z 354.28,A -85,B 0,C 180,E1 -12209.687,E2 -12209.687} C_VEL
LIN {X 0,Y 376.001,Z 354.263,A -85,B 0,C 180,E1 -12212.142,E2 -12212.142} C_VEL
LIN {X 0,Y 376.005,Z 354.268,A -85,B 0,C 180,E1 -12214.539,E2 -12214.539} C_VEL
LIN {X 0,Y 375.961,Z 354.271,A -85,B 0,C 180,E1 -12218.045,E2 -12218.045} C_VEL
LIN {X 0,Y 376.007,Z 354.267,A -85,B 0,C 180,E1 -12221.473,E2 -12221.473} C_VEL
LIN {X 0,Y 376.058,Z 354.261,A -85,B 0,C 180,E1 -12224.832,E2 -12224.832} C_VEL
LIN {X 0,Y 376.057,Z 354.253,A -85,B 0,C 180,E1 -12228.137,E2 -12228.137} C_VEL
LIN {X 0,Y 376.256,Z 354.24,A -85,B 0,C 180,E1 -12231.877,E2 -12231.877} C_VEL
LIN {X 0,Y 376.17,Z 354.253,A -85,B 0,C 180,E1 -12234.64,E2 -12234.64} C_VEL
LIN {X 0,Y 376.352,Z 354.23,A -85,B 0,C 180,E1 -12237.86,E2 -12237.86} C_VEL
LIN {X 0,Y 376.487,Z 354.216,A -85,B 0,C 180,E1 -12240,E2 -12240} C_VEL
LIN {X 0,Y 376.189,Z 354.253,A -85,B 0,C 180,E1 -12243.213,E2 -12243.213} C_VEL
LIN {X 0,Y 376.245,Z 354.245,A -85,B 0,C 180,E1 -12246.435,E2 -12246.435} C_VEL
LIN {X 0,Y 376.203,Z 354.248,A -85,B 0,C 180,E1 -12248.595,E2 -12248.595} C_VEL
LIN {X 0,Y 376.048,Z 354.267,A -85,B 0,C 180,E1 -12251.863,E2 -12251.863} C_VEL
LIN {X 0,Y 376.056,Z 354.266,A -85,B 0,C 180,E1 -12255.167,E2 -12255.167} C_VEL
LIN {X 0,Y 376.021,Z 354.27,A -85,B 0,C 180,E1 -12258.526,E2 -12258.526} C_VEL
LIN {X 0,Y 375.961,Z 354.28,A -85,B 0,C 180,E1 -12261.954,E2 -12261.954} C_VEL
LIN {X 0,Y 376.004,Z 354.275,A -85,B 0,C 180,E1 -12265.461,E2 -12265.461} C_VEL
LIN {X 0,Y 375.974,Z 354.281,A -85,B 0,C 180,E1 -12269.079,E2 -12269.079} C_VEL
LIN {X 0,Y 375.949,Z 354.282,A -85,B 0,C 180,E1 -12272.828,E2 -12272.828} C_VEL
LIN {X 0,Y 375.956,Z 354.28,A -85,B 0,C 180,E1 -12275.416,E2 -12275.416} C_VEL
LIN {X 0,Y 375.968,Z 354.423,A -85,B 0,C 180,E1 -12277.242,E2 -12277.242} C_VEL
LIN {X 0,Y 376.582,Z 357.897,A -85,B 0,C 180,E1 -12280.079,E2 -12280.079} C_VEL
LIN {X 0,Y 377.363,Z 362.518,A -85,B 0,C 180,E1 -12283.558,E2 -12283.558} C_VEL
LIN {X 0,Y 378.035,Z 366.782,A -85,B 0,C 180,E1 -12286.54,E2 -12286.54} C_VEL
LIN {X 0,Y 378.182,Z 370.124,A -85,B 0,C 180,E1 -12288.722,E2 -12288.722} C_VEL
LIN {X 0,Y 377.6,Z 375.694,A -85,B 0,C 180,E1 -12292.106,E2 -12292.106} C_VEL
LIN {X 0,Y 377.16,Z 380.771,A -85,B 0,C 180,E1 -12295.074,E2 -12295.074} C_VEL
LIN {X 0,Y 376.613,Z 386.796,A -85,B 0,C 180,E1 -12298.5,E2 -12298.5} C_VEL
LIN {X 0,Y 375.96,Z 393.297,A -85,B 0,C 180,E1 -12302.139,E2 -12302.139} C_VEL
LIN {X 0,Y 375.916,Z 393.977,A -85,B 0,C 180,E1 -12302.518,E2 -12302.518} C_VEL
LIN {X 0,Y 378.585,Z 403.077,A -85,B 0,C 180,E1 -12302.946,E2 -12302.946} C_VEL
LIN {X 0,Y 382.435,Z 418.096,A -85,B 0,C 180,E1 -12303.761,E2 -12303.761} C_VEL
LIN {X 0,Y 385.133,Z 431.513,A -85,B 0,C 180,E1 -12304.61,E2 -12304.61} C_VEL
LIN {X 0,Y 386.641,Z 442.66,A -85,B 0,C 180,E1 -12305.39,E2 -12305.39} C_VEL
LIN {X 0,Y 385.253,Z 456.355,A -85,B 0,C 180,E1 -12306.339,E2 -12306.339} C_VEL
LIN {X 0,Y 383.51,Z 469.992,A -85,B 0,C 180,E1 -12307.509,E2 -12307.509} C_VEL
LIN {X 0,Y 381.669,Z 483.617,A -85,B 0,C 180,E1 -12308.957,E2 -12308.957} C_VEL
LIN {X 0,Y 380.014,Z 495.889,A -85,B 0,C 180,E1 -12310.556,E2 -12310.556} C_VEL
LIN {X 0,Y 378.669,Z 506.2,A -85,B 0,C 180,E1 -12312.168,E2 -12312.168} C_VEL
LIN {X 0,Y 377.253,Z 516.283,A -85,B 0,C 180,E1 -12314.051,E2 -12314.051} C_VEL
LIN {X 0,Y 376.231,Z 524.67,A -85,B 0,C 180,E1 -12315.946,E2 -12315.946} C_VEL
LIN {X 0,Y 375.465,Z 532.563,A -85,B 0,C 180,E1 -12318.118,E2 -12318.118} C_VEL
LIN {X 0,Y 374.886,Z 538.846,A -85,B 0,C 180,E1 -12320.287,E2 -12320.287} C_VEL
LIN {X 0,Y 374.652,Z 543.717,A -85,B 0,C 180,E1 -12322.455,E2 -12322.455} C_VEL
LIN {X 0,Y 374.535,Z 547.288,A -85,B 0,C 180,E1 -12324.617,E2 -12324.617} C_VEL
LIN {X 0,Y 374.494,Z 549.638,A -85,B 0,C 180,E1 -12326.773,E2 -12326.773} C_VEL
LIN {X 0,Y 374.621,Z 550.827,A -85,B 0,C 180,E1 -12328.926,E2 -12328.926} C_VEL
LIN {X 0,Y 374.621,Z 550.825,A -85,B 0,C 180,E1 -12331.075,E2 -12331.075} C_VEL
LIN {X 0,Y 374.496,Z 549.629,A -85,B 0,C 180,E1 -12333.228,E2 -12333.228} C_VEL
LIN {X 0,Y 374.574,Z 547.275,A -85,B 0,C 180,E1 -12335.383,E2 -12335.383} C_VEL
LIN {X 0,Y 374.633,Z 545.647,A -85,B 0,C 180,E1 -12336.463,E2 -12336.463} C_VEL
LIN {X 0,Y 374.75,Z 541.436,A -85,B 0,C 180,E1 -12338.629,E2 -12338.629} C_VEL
LIN {X 0,Y 375.111,Z 535.866,A -85,B 0,C 180,E1 -12340.799,E2 -12340.799} C_VEL
LIN {X 0,Y 375.827,Z 528.795,A -85,B 0,C 180,E1 -12342.968,E2 -12342.968} C_VEL
LIN {X 0,Y 376.785,Z 520.002,A -85,B 0,C 180,E1 -12345.138,E2 -12345.138} C_VEL
LIN {X 0,Y 377.941,Z 510.674,A -85,B 0,C 180,E1 -12347.031,E2 -12347.031} C_VEL
LIN {X 0,Y 379.457,Z 499.913,A -85,B 0,C 180,E1 -12348.837,E2 -12348.837} C_VEL
LIN {X 0,Y 381.067,Z 487.859,A -85,B 0,C 180,E1 -12350.513,E2 -12350.513} C_VEL
LIN {X 0,Y 382.817,Z 475.138,A -85,B 0,C 180,E1 -12351.967,E2 -12351.967} C_VEL
LIN {X 0,Y 384.457,Z 462.624,A -85,B 0,C 180,E1 -12353.143,E2 -12353.143} C_VEL
LIN {X 0,Y 386.048,Z 448.513,A -85,B 0,C 180,E1 -12354.22,E2 -12354.22} C_VEL
LIN {X 0,Y 386.649,Z 441.822,A -85,B 0,C 180,E1 -12354.656,E2 -12354.656} C_VEL
LIN {X 0,Y 384.256,Z 426.729,A -85,B 0,C 180,E1 -12355.701,E2 -12355.701} C_VEL
LIN {X 0,Y 380.804,Z 411.229,A -85,B 0,C 180,E1 -12356.618,E2 -12356.618} C_VEL
LIN {X 0,Y 376.581,Z 396.706,A -85,B 0,C 180,E1 -12357.353,E2 -12357.353} C_VEL
LIN {X 0,Y 375.948,Z 393.972,A -85,B 0,C 180,E1 -12357.472,E2 -12357.472} C_VEL
LIN {X 0,Y 376.452,Z 387.991,A -85,B 0,C 180,E1 -12360.821,E2 -12360.821} C_VEL
LIN {X 0,Y 376.981,Z 382.305,A -85,B 0,C 180,E1 -12364.007,E2 -12364.007} C_VEL
LIN {X 0,Y 377.429,Z 377.524,A -85,B 0,C 180,E1 -12366.804,E2 -12366.804} C_VEL
LIN {X 0,Y 378.047,Z 371.157,A -85,B 0,C 180,E1 -12370.592,E2 -12370.592} C_VEL
LIN {X 0,Y 378.115,Z 367.791,A -85,B 0,C 180,E1 -12372.721,E2 -12372.721} C_VEL
LIN {X 0,Y 377.548,Z 363.427,A -85,B 0,C 180,E1 -12375.729,E2 -12375.729} C_VEL
LIN {X 0,Y 376.715,Z 358.712,A -85,B 0,C 180,E1 -12379.235,E2 -12379.235} C_VEL
LIN {X 0,Y 376.031,Z 354.572,A -85,B 0,C 180,E1 -12382.597,E2 -12382.597} C_VEL
LIN {X 0,Y 375.957,Z 354.284,A -85,B 0,C 180,E1 -12383.259,E2 -12383.259} C_VEL
LIN {X 0,Y 375.962,Z 354.281,A -85,B 0,C 180,E1 -12385.889,E2 -12385.889} C_VEL
LIN {X 0,Y 375.967,Z 354.278,A -85,B 0,C 180,E1 -12389.688,E2 -12389.688} C_VEL
LIN {X 0,Y 376.022,Z 354.272,A -85,B 0,C 180,E1 -12393.348,E2 -12393.348} C_VEL
LIN {X 0,Y 375.999,Z 354.277,A -85,B 0,C 180,E1 -12396.889,E2 -12396.889} C_VEL
LIN {X 0,Y 376.001,Z 354.275,A -85,B 0,C 180,E1 -12400.34,E2 -12400.34} C_VEL
LIN {X 0,Y 376.032,Z 354.272,A -85,B 0,C 180,E1 -12403.719,E2 -12403.719} C_VEL
LIN {X 0,Y 376.107,Z 354.264,A -85,B 0,C 180,E1 -12407.042,E2 -12407.042} C_VEL
LIN {X 0,Y 376.122,Z 354.262,A -85,B 0,C 180,E1 -12410.319,E2 -12410.319} C_VEL
LIN {X 0,Y 376.234,Z 354.247,A -85,B 0,C 180,E1 -12412.487,E2 -12412.487} C_VEL
LIN {X 0,Y 376.175,Z 354.252,A -85,B 0,C 180,E1 -12414.64,E2 -12414.64} C_VEL
LIN {X 0,Y 376.357,Z 354.229,A -85,B 0,C 180,E1 -12417.86,E2 -12417.86} C_VEL
LIN {X 0,Y 376.491,Z 354.212,A -85,B 0,C 180,E1 -12420,E2 -12420} C_VEL
LIN {X 0,Y 376.192,Z 354.247,A -85,B 0,C 180,E1 -12423.213,E2 -12423.213} C_VEL
LIN {X 0,Y 376.239,Z 354.24,A -85,B 0,C 180,E1 -12426.612,E2 -12426.612} C_VEL
LIN {X 0,Y 376.209,Z 354.248,A -85,B 0,C 180,E1 -12428.595,E2 -12428.595} C_VEL
LIN {X 0,Y 376.053,Z 354.249,A -85,B 0,C 180,E1 -12431.863,E2 -12431.863} C_VEL
LIN {X 0,Y 376.062,Z 354.262,A -85,B 0,C 180,E1 -12435.167,E2 -12435.167} C_VEL
LIN {X 0,Y 376.012,Z 354.265,A -85,B 0,C 180,E1 -12438.527,E2 -12438.527} C_VEL
LIN {X 0,Y 375.961,Z 354.271,A -85,B 0,C 180,E1 -12441.955,E2 -12441.955} C_VEL
LIN {X 0,Y 376.009,Z 354.269,A -85,B 0,C 180,E1 -12445.461,E2 -12445.461} C_VEL
LIN {X 0,Y 375.964,Z 354.275,A -85,B 0,C 180,E1 -12449.08,E2 -12449.08} C_VEL
LIN {X 0,Y 375.952,Z 354.27,A -85,B 0,C 180,E1 -12452.828,E2 -12452.828} C_VEL
LIN {X 0,Y 375.961,Z 354.278,A -85,B 0,C 180,E1 -12455.415,E2 -12455.415} C_VEL
LIN {X 0,Y 375.979,Z 354.278,A -85,B 0,C 180,E1 -12458.271,E2 -12458.271} C_VEL
LIN {X 0,Y 375.937,Z 354.283,A -85,B 0,C 180,E1 -12461.601,E2 -12461.601} C_VEL
LIN {X 0,Y 375.929,Z 354.288,A -85,B 0,C 180,E1 -12465.269,E2 -12465.269} C_VEL
LIN {X 0,Y 375.863,Z 354.296,A -85,B 0,C 180,E1 -12468.412,E2 -12468.412} C_VEL
LIN {X 0,Y 375.694,Z 354.315,A -85,B 0,C 180,E1 -12470.503,E2 -12470.503} C_VEL
LIN {X 0,Y 375.594,Z 354.594,A -85,B 0,C 180,E1 -12471.867,E2 -12471.867} C_VEL
LIN {X 0,Y 375.5,Z 357.293,A -85,B 0,C 180,E1 -12475.439,E2 -12475.439} C_VEL
LIN {X 0,Y 375.386,Z 359.642,A -85,B 0,C 180,E1 -12478.384,E2 -12478.384} C_VEL
LIN {X 0,Y 375.275,Z 362.428,A -85,B 0,C 180,E1 -12481.666,E2 -12481.666} C_VEL
LIN {X 0,Y 375.236,Z 363.233,A -85,B 0,C 180,E1 -12482.567,E2 -12482.567} C_VEL
LIN {X 0,Y 376.297,Z 366.354,A -85,B 0,C 180,E1 -12482.73,E2 -12482.73} C_VEL
LIN {X 0,Y 382.068,Z 381.251,A -85,B 0,C 180,E1 -12483.659,E2 -12483.659} C_VEL
LIN {X 0,Y 386.491,Z 395.528,A -85,B 0,C 180,E1 -12484.66,E2 -12484.66} C_VEL
LIN {X 0,Y 388.193,Z 402.298,A -85,B 0,C 180,E1 -12485.175,E2 -12485.175} C_VEL
LIN {X 0,Y 386.97,Z 416.446,A -85,B 0,C 180,E1 -12486.08,E2 -12486.08} C_VEL
LIN {X 0,Y 385.626,Z 428.954,A -85,B 0,C 180,E1 -12487.073,E2 -12487.073} C_VEL
LIN {X 0,Y 383.947,Z 442.381,A -85,B 0,C 180,E1 -12488.384,E2 -12488.384} C_VEL
LIN {X 0,Y 382.387,Z 454.074,A -85,B 0,C 180,E1 -12489.776,E2 -12489.776} C_VEL
LIN {X 0,Y 380.785,Z 465.627,A -85,B 0,C 180,E1 -12491.435,E2 -12491.435} C_VEL
LIN {X 0,Y 379.198,Z 476.38,A -85,B 0,C 180,E1 -12493.305,E2 -12493.305} C_VEL
LIN {X 0,Y 377.81,Z 485.82,A -85,B 0,C 180,E1 -12495.308,E2 -12495.308} C_VEL
LIN {X 0,Y 376.975,Z 492.671,A -85,B 0,C 180,E1 -12497.072,E2 -12497.072} C_VEL
LIN {X 0,Y 375.983,Z 499.571,A -85,B 0,C 180,E1 -12499.226,E2 -12499.226} C_VEL
LIN {X 0,Y 375.399,Z 504.982,A -85,B 0,C 180,E1 -12501.386,E2 -12501.386} C_VEL
LIN {X 0,Y 374.992,Z 509.065,A -85,B 0,C 180,E1 -12503.543,E2 -12503.543} C_VEL
LIN {X 0,Y 374.719,Z 511.934,A -85,B 0,C 180,E1 -12505.697,E2 -12505.697} C_VEL
LIN {X 0,Y 374.74,Z 513.651,A -85,B 0,C 180,E1 -12507.85,E2 -12507.85} C_VEL
LIN {X 0,Y 374.615,Z 514.258,A -85,B 0,C 180,E1 -12510,E2 -12510} C_VEL
LIN {X 0,Y 374.74,Z 513.697,A -85,B 0,C 180,E1 -12512.149,E2 -12512.149} C_VEL
LIN {X 0,Y 374.717,Z 512.04,A -85,B 0,C 180,E1 -12514.302,E2 -12514.302} C_VEL
LIN {X 0,Y 375.003,Z 508.922,A -85,B 0,C 180,E1 -12516.644,E2 -12516.644} C_VEL
LIN {X 0,Y 375.374,Z 505.202,A -85,B 0,C 180,E1 -12518.614,E2 -12518.614} C_VEL
LIN {X 0,Y 375.956,Z 499.86,A -85,B 0,C 180,E1 -12520.774,E2 -12520.774} C_VEL
LIN {X 0,Y 376.915,Z 493.041,A -85,B 0,C 180,E1 -12522.929,E2 -12522.929} C_VEL
LIN {X 0,Y 377.978,Z 484.531,A -85,B 0,C 180,E1 -12525.088,E2 -12525.088} C_VEL
LIN {X 0,Y 379.314,Z 475.468,A -85,B 0,C 180,E1 -12526.966,E2 -12526.966} C_VEL
LIN {X 0,Y 380.698,Z 466.224,A -85,B 0,C 180,E1 -12528.569,E2 -12528.569} C_VEL
LIN {X 0,Y 382.318,Z 454.375,A -85,B 0,C 180,E1 -12530.286,E2 -12530.286} C_VEL
LIN {X 0,Y 384.004,Z 442.03,A -85,B 0,C 180,E1 -12531.753,E2 -12531.753} C_VEL
LIN {X 0,Y 385.677,Z 428.523,A -85,B 0,C 180,E1 -12533.065,E2 -12533.065} C_VEL
LIN {X 0,Y 387.079,Z 415.727,A -85,B 0,C 180,E1 -12534.072,E2 -12534.072} C_VEL
LIN {X 0,Y 387.63,Z 408.98,A -85,B 0,C 180,E1 -12534.528,E2 -12534.528} C_VEL
LIN {X 0,Y 387.204,Z 405.595,A -85,B 0,C 180,E1 -12534.796,E2 -12534.796} C_VEL
LIN {X 0,Y 385.586,Z 402.636,A -85,B 0,C 180,E1 -12535.108,E2 -12535.108} C_VEL
LIN {X 0,Y 380.351,Z 396.267,A -85,B 0,C 180,E1 -12535.867,E2 -12535.867} C_VEL
LIN {X 0,Y 378.774,Z 392.979,A -85,B 0,C 180,E1 -12536.161,E2 -12536.161} C_VEL
LIN {X 0,Y 374.698,Z 380.394,A -85,B 0,C 180,E1 -12537.056,E2 -12537.056} C_VEL
LIN {X 0,Y 369.028,Z 366.268,A -85,B 0,C 180,E1 -12537.971,E2 -12537.971} C_VEL
LIN {X 0,Y 368.209,Z 363.529,A -85,B 0,C 180,E1 -12538.132,E2 -12538.132} C_VEL
LIN {X 0,Y 368.307,Z 361.1,A -85,B 0,C 180,E1 -12541.011,E2 -12541.011} C_VEL
LIN {X 0,Y 368.417,Z 359.074,A -85,B 0,C 180,E1 -12543.587,E2 -12543.587} C_VEL
LIN {X 0,Y 368.483,Z 356.632,A -85,B 0,C 180,E1 -12546.769,E2 -12546.769} C_VEL
LIN {X 0,Y 368.575,Z 355.201,A -85,B 0,C 180,E1 -12548.994,E2 -12548.994} C_VEL
LIN {X 0,Y 368.821,Z 355.165,A -85,B 0,C 180,E1 -12551.999,E2 -12551.999} C_VEL
LIN {X 0,Y 368.878,Z 355.161,A -85,B 0,C 180,E1 -12555.175,E2 -12555.175} C_VEL
LIN {X 0,Y 368.881,Z 355.161,A -85,B 0,C 180,E1 -12558.177,E2 -12558.177} C_VEL
LIN {X 0,Y 368.909,Z 355.156,A -85,B 0,C 180,E1 -12561.359,E2 -12561.359} C_VEL
LIN {X 0,Y 368.935,Z 355.153,A -85,B 0,C 180,E1 -12565.146,E2 -12565.146} C_VEL
LIN {X 0,Y 368.927,Z 355.154,A -85,B 0,C 180,E1 -12569.046,E2 -12569.046} C_VEL
LIN {X 0,Y 368.985,Z 355.14,A -85,B 0,C 180,E1 -12571.564,E2 -12571.564} C_VEL
LIN {X 0,Y 368.956,Z 355.149,A -85,B 0,C 180,E1 -12575.224,E2 -12575.224} C_VEL
LIN {X 0,Y 368.935,Z 355.136,A -85,B 0,C 180,E1 -12578.973,E2 -12578.973} C_VEL
LIN {X 0,Y 368.988,Z 355.148,A -85,B 0,C 180,E1 -12582.257,E2 -12582.257} C_VEL
LIN {X 0,Y 369.035,Z 355.123,A -85,B 0,C 180,E1 -12586.227,E2 -12586.227} C_VEL
LIN {X 0,Y 369.07,Z 355.137,A -85,B 0,C 180,E1 -12590.132,E2 -12590.132} C_VEL
LIN {X 0,Y 369.186,Z 355.122,A -85,B 0,C 180,E1 -12592.342,E2 -12592.342} C_VEL
LIN {X 0,Y 369.143,Z 355.129,A -85,B 0,C 180,E1 -12594.537,E2 -12594.537} C_VEL
LIN {X 0,Y 369.317,Z 355.106,A -85,B 0,C 180,E1 -12597.819,E2 -12597.819} C_VEL
LIN {X 0,Y 369.456,Z 355.092,A -85,B 0,C 180,E1 -12600,E2 -12600} C_VEL
LIN {X 0,Y 369.317,Z 355.106,A -85,B 0,C 180,E1 -12602.181,E2 -12602.181} C_VEL
LIN {X 0,Y 369.206,Z 355.122,A -85,B 0,C 180,E1 -12606.558,E2 -12606.558} C_VEL
LIN {X 0,Y 369.135,Z 355.129,A -85,B 0,C 180,E1 -12608.761,E2 -12608.761} C_VEL
LIN {X 0,Y 369.004,Z 355.144,A -85,B 0,C 180,E1 -12612.093,E2 -12612.093} C_VEL
LIN {X 0,Y 368.995,Z 355.144,A -85,B 0,C 180,E1 -12615.465,E2 -12615.465} C_VEL
LIN {X 0,Y 368.98,Z 355.149,A -85,B 0,C 180,E1 -12618.893,E2 -12618.893} C_VEL
LIN {X 0,Y 368.93,Z 355.155,A -85,B 0,C 180,E1 -12622.395,E2 -12622.395} C_VEL
LIN {X 0,Y 368.997,Z 355.151,A -85,B 0,C 180,E1 -12625.98,E2 -12625.98} C_VEL
LIN {X 0,Y 368.965,Z 355.154,A -85,B 0,C 180,E1 -12628.814,E2 -12628.814} C_VEL
LIN {X 0,Y 368.898,Z 355.158,A -85,B 0,C 180,E1 -12632.238,E2 -12632.238} C_VEL
LIN {X 0,Y 368.927,Z 355.156,A -85,B 0,C 180,E1 -12635.002,E2 -12635.002} C_VEL
LIN {X 0,Y 368.943,Z 355.334,A -85,B 0,C 180,E1 -12636.763,E2 -12636.763} C_VEL
LIN {X 0,Y 369.673,Z 359.535,A -85,B 0,C 180,E1 -12640.27,E2 -12640.27} C_VEL
LIN {X 0,Y 370.488,Z 364.266,A -85,B 0,C 180,E1 -12643.877,E2 -12643.877} C_VEL
LIN {X 0,Y 371.097,Z 368.722,A -85,B 0,C 180,E1 -12647.018,E2 -12647.018} C_VEL
LIN {X 0,Y 371.097,Z 372.136,A -85,B 0,C 180,E1 -12649.247,E2 -12649.247} C_VEL
LIN {X 0,Y 370.455,Z 377.953,A -85,B 0,C 180,E1 -12652.825,E2 -12652.825} C_VEL
LIN {X 0,Y 369.971,Z 383.159,A -85,B 0,C 180,E1 -12655.918,E2 -12655.918} C_VEL
LIN {X 0,Y 369.337,Z 389.713,A -85,B 0,C 180,E1 -12659.718,E2 -12659.718} C_VEL
LIN {X 0,Y 368.912,Z 393.605,A -85,B 0,C 180,E1 -12661.95,E2 -12661.95} C_VEL
LIN {X 0,Y 369.785,Z 396.883,A -85,B 0,C 180,E1 -12662.101,E2 -12662.101} C_VEL
LIN {X 0,Y 373.943,Z 411.099,A -85,B 0,C 180,E1 -12662.851,E2 -12662.851} C_VEL
LIN {X 0,Y 377.441,Z 426.426,A -85,B 0,C 180,E1 -12663.793,E2 -12663.793} C_VEL
LIN {X 0,Y 379.751,Z 440.718,A -85,B 0,C 180,E1 -12664.808,E2 -12664.808} C_VEL
LIN {X 0,Y 379.922,Z 444.844,A -85,B 0,C 180,E1 -12665.11,E2 -12665.11} C_VEL
LIN {X 0,Y 378.308,Z 459.221,A -85,B 0,C 180,E1 -12666.168,E2 -12666.168} C_VEL
LIN {X 0,Y 376.561,Z 472.279,A -85,B 0,C 180,E1 -12667.361,E2 -12667.361} C_VEL
LIN {X 0,Y 374.822,Z 484.347,A -85,B 0,C 180,E1 -12668.698,E2 -12668.698} C_VEL
LIN {X 0,Y 373.272,Z 495.54,A -85,B 0,C 180,E1 -12670.19,E2 -12670.19} C_VEL
LIN {X 0,Y 371.833,Z 505.85,A -85,B 0,C 180,E1 -12671.829,E2 -12671.829} C_VEL
LIN {X 0,Y 370.34,Z 515.932,A -85,B 0,C 180,E1 -12673.745,E2 -12673.745} C_VEL
LIN {X 0,Y 369.264,Z 524.32,A -85,B 0,C 180,E1 -12675.676,E2 -12675.676} C_VEL
LIN {X 0,Y 368.423,Z 532.211,A -85,B 0,C 180,E1 -12677.888,E2 -12677.888} C_VEL
LIN {X 0,Y 367.811,Z 538.495,A -85,B 0,C 180,E1 -12680.098,E2 -12680.098} C_VEL
LIN {X 0,Y 367.573,Z 543.368,A -85,B 0,C 180,E1 -12682.309,E2 -12682.309} C_VEL
LIN {X 0,Y 367.451,Z 546.94,A -85,B 0,C 180,E1 -12684.513,E2 -12684.513} C_VEL
LIN {X 0,Y 367.409,Z 549.291,A -85,B 0,C 180,E1 -12686.711,E2 -12686.711} C_VEL
LIN {X 0,Y 367.554,Z 550.481,A -85,B 0,C 180,E1 -12688.905,E2 -12688.905} C_VEL
LIN {X 0,Y 367.554,Z 550.479,A -85,B 0,C 180,E1 -12691.096,E2 -12691.096} C_VEL
LIN {X 0,Y 367.411,Z 549.281,A -85,B 0,C 180,E1 -12693.29,E2 -12693.29} C_VEL
LIN {X 0,Y 367.492,Z 546.926,A -85,B 0,C 180,E1 -12695.488,E2 -12695.488} C_VEL
LIN {X 0,Y 367.576,Z 543.352,A -85,B 0,C 180,E1 -12697.692,E2 -12697.692} C_VEL
LIN {X 0,Y 367.812,Z 538.476,A -85,B 0,C 180,E1 -12699.903,E2 -12699.903} C_VEL
LIN {X 0,Y 368.428,Z 532.178,A -85,B 0,C 180,E1 -12702.113,E2 -12702.113} C_VEL
LIN {X 0,Y 369.266,Z 524.275,A -85,B 0,C 180,E1 -12704.325,E2 -12704.325} C_VEL
LIN {X 0,Y 370.343,Z 515.883,A -85,B 0,C 180,E1 -12706.255,E2 -12706.255} C_VEL
LIN {X 0,Y 371.791,Z 505.789,A -85,B 0,C 180,E1 -12708.174,E2 -12708.174} C_VEL
LIN {X 0,Y 373.273,Z 495.475,A -85,B 0,C 180,E1 -12709.811,E2 -12709.811} C_VEL
LIN {X 0,Y 375.042,Z 483.197,A -85,B 0,C 180,E1 -12711.434,E2 -12711.434} C_VEL
LIN {X 0,Y 376.885,Z 469.538,A -85,B 0,C 180,E1 -12712.909,E2 -12712.909} C_VEL
LIN {X 0,Y 378.737,Z 455.862,A -85,B 0,C 180,E1 -12714.095,E2 -12714.095} C_VEL
LIN {X 0,Y 380.005,Z 442.964,A -85,B 0,C 180,E1 -12715.011,E2 -12715.011} C_VEL
LIN {X 0,Y 378.049,Z 429.856,A -85,B 0,C 180,E1 -12715.962,E2 -12715.962} C_VEL
LIN {X 0,Y 374.758,Z 414.394,A -85,B 0,C 180,E1 -12716.942,E2 -12716.942} C_VEL
LIN {X 0,Y 370.763,Z 399.915,A -85,B 0,C 180,E1 -12717.73,E2 -12717.73} C_VEL
LIN {X 0,Y 369.023,Z 394.318,A -85,B 0,C 180,E1 -12718.007,E2 -12718.007} C_VEL
LIN {X 0,Y 368.938,Z 393.534,A -85,B 0,C 180,E1 -12718.076,E2 -12718.076} C_VEL
LIN {X 0,Y 369.428,Z 388.249,A -85,B 0,C 180,E1 -12721.121,E2 -12721.121} C_VEL
LIN {X 0,Y 370.061,Z 381.985,A -85,B 0,C 180,E1 -12724.733,E2 -12724.733} C_VEL
LIN {X 0,Y 370.585,Z 376.473,A -85,B 0,C 180,E1 -12728.051,E2 -12728.051} C_VEL
LIN {X 0,Y 371.166,Z 370.848,A -85,B 0,C 180,E1 -12731.508,E2 -12731.508} C_VEL
LIN {X 0,Y 370.936,Z 367.212,A -85,B 0,C 180,E1 -12733.948,E2 -12733.948} C_VEL
LIN {X 0,Y 370.289,Z 363.14,A -85,B 0,C 180,E1 -12736.9,E2 -12736.9} C_VEL
LIN {X 0,Y 369.679,Z 359.45,A -85,B 0,C 180,E1 -12739.731,E2 -12739.731} C_VEL
LIN {X 0,Y 368.939,Z 355.295,A -85,B 0,C 180,E1 -12743.237,E2 -12743.237} C_VEL
LIN {X 0,Y 368.899,Z 355.163,A -85,B 0,C 180,E1 -12746.462,E2 -12746.462} C_VEL
LIN {X 0,Y 368.931,Z 355.154,A -85,B 0,C 180,E1 -12749.047,E2 -12749.047} C_VEL
LIN {X 0,Y 368.965,Z 355.152,A -85,B 0,C 180,E1 -12752.797,E2 -12752.797} C_VEL
LIN {X 0,Y 368.948,Z 355.153,A -85,B 0,C 180,E1 -12756.113,E2 -12756.113} C_VEL
LIN {X 0,Y 368.94,Z 355.156,A -85,B 0,C 180,E1 -12759.947,E2 -12759.947} C_VEL
LIN {X 0,Y 368.979,Z 355.152,A -85,B 0,C 180,E1 -12763.399,E2 -12763.399} C_VEL
LIN {X 0,Y 369.061,Z 355.141,A -85,B 0,C 180,E1 -12766.79,E2 -12766.79} C_VEL
LIN {X 0,Y 369.071,Z 355.14,A -85,B 0,C 180,E1 -12770.132,E2 -12770.132} C_VEL
LIN {X 0,Y 369.192,Z 355.126,A -85,B 0,C 180,E1 -12772.342,E2 -12772.342} C_VEL
LIN {X 0,Y 369.148,Z 355.128,A -85,B 0,C 180,E1 -12774.538,E2 -12774.538} C_VEL
LIN {X 0,Y 369.322,Z 355.105,A -85,B 0,C 180,E1 -12777.819,E2 -12777.819} C_VEL
LIN {X 0,Y 369.46,Z 355.087,A -85,B 0,C 180,E1 -12780,E2 -12780} C_VEL
LIN {X 0,Y 369.322,Z 355.105,A -85,B 0,C 180,E1 -12782.181,E2 -12782.181} C_VEL
LIN {X 0,Y 369.209,Z 355.115,A -85,B 0,C 180,E1 -12786.6,E2 -12786.6} C_VEL
LIN {X 0,Y 369.141,Z 355.13,A -85,B 0,C 180,E1 -12788.761,E2 -12788.761} C_VEL
LIN {X 0,Y 369.008,Z 355.123,A -85,B 0,C 180,E1 -12792.093,E2 -12792.093} C_VEL
LIN {X 0,Y 369.001,Z 355.144,A -85,B 0,C 180,E1 -12795.465,E2 -12795.465} C_VEL
LIN {X 0,Y 368.962,Z 355.142,A -85,B 0,C 180,E1 -12798.894,E2 -12798.894} C_VEL
LIN {X 0,Y 368.928,Z 355.148,A -85,B 0,C 180,E1 -12802.396,E2 -12802.396} C_VEL
LIN {X 0,Y 369.003,Z 355.136,A -85,B 0,C 180,E1 -12805.98,E2 -12805.98} C_VEL
LIN {X 0,Y 368.918,Z 355.154,A -85,B 0,C 180,E1 -12809.69,E2 -12809.69} C_VEL
LIN {X 0,Y 368.9,Z 355.146,A -85,B 0,C 180,E1 -12813.043,E2 -12813.043} C_VEL
LIN {X 0,Y 368.921,Z 355.157,A -85,B 0,C 180,E1 -12816.196,E2 -12816.196} C_VEL
LIN {X 0,Y 368.908,Z 355.158,A -85,B 0,C 180,E1 -12818.953,E2 -12818.953} C_VEL
LIN {X 0,Y 368.884,Z 355.162,A -85,B 0,C 180,E1 -12822.009,E2 -12822.009} C_VEL
LIN {X 0,Y 368.882,Z 355.165,A -85,B 0,C 180,E1 -12825.176,E2 -12825.176} C_VEL
LIN {X 0,Y 368.82,Z 355.173,A -85,B 0,C 180,E1 -12828.168,E2 -12828.168} C_VEL
LIN {X 0,Y 368.532,Z 355.221,A -85,B 0,C 180,E1 -12831.433,E2 -12831.433} C_VEL
LIN {X 0,Y 368.45,Z 357.958,A -85,B 0,C 180,E1 -12835.105,E2 -12835.105} C_VEL
LIN {X 0,Y 368.371,Z 359.984,A -85,B 0,C 180,E1 -12837.71,E2 -12837.71} C_VEL
LIN {X 0,Y 368.236,Z 363.139,A -85,B 0,C 180,E1 -12841.501,E2 -12841.501} C_VEL
LIN {X 0,Y 368.255,Z 363.564,A -85,B 0,C 180,E1 -12841.994,E2 -12841.994} C_VEL
LIN {X 0,Y 369.269,Z 366.666,A -85,B 0,C 180,E1 -12842.164,E2 -12842.164} C_VEL
LIN {X 0,Y 374.919,Z 380.966,A -85,B 0,C 180,E1 -12843.088,E2 -12843.088} C_VEL
LIN {X 0,Y 378.981,Z 393.538,A -85,B 0,C 180,E1 -12843.984,E2 -12843.984} C_VEL
LIN {X 0,Y 381.508,Z 403.019,A -85,B 0,C 180,E1 -12844.733,E2 -12844.733} C_VEL
LIN {X 0,Y 381.473,Z 406.062,A -85,B 0,C 180,E1 -12844.929,E2 -12844.929} C_VEL
LIN {X 0,Y 380.159,Z 419.929,A -85,B 0,C 180,E1 -12845.883,E2 -12845.883} C_VEL
LIN {X 0,Y 378.75,Z 432.149,A -85,B 0,C 180,E1 -12846.921,E2 -12846.921} C_VEL
LIN {X 0,Y 377.021,Z 445.063,A -85,B 0,C 180,E1 -12848.254,E2 -12848.254} C_VEL
LIN {X 0,Y 375.261,Z 457.579,A -85,B 0,C 180,E1 -12849.837,E2 -12849.837} C_VEL
LIN {X 0,Y 373.523,Z 469.217,A -85,B 0,C 180,E1 -12851.629,E2 -12851.629} C_VEL
LIN {X 0,Y 371.955,Z 479.408,A -85,B 0,C 180,E1 -12853.535,E2 -12853.535} C_VEL
LIN {X 0,Y 370.606,Z 487.86,A -85,B 0,C 180,E1 -12855.446,E2 -12855.446} C_VEL
LIN {X 0,Y 369.693,Z 494.886,A -85,B 0,C 180,E1 -12857.372,E2 -12857.372} C_VEL
LIN {X 0,Y 368.8,Z 501.401,A -85,B 0,C 180,E1 -12859.569,E2 -12859.569} C_VEL
LIN {X 0,Y 368.254,Z 506.485,A -85,B 0,C 180,E1 -12861.77,E2 -12861.77} C_VEL
LIN {X 0,Y 367.921,Z 509.414,A -85,B 0,C 180,E1 -12863.418,E2 -12863.418} C_VEL
LIN {X 0,Y 367.65,Z 512.282,A -85,B 0,C 180,E1 -12865.614,E2 -12865.614} C_VEL
LIN {X 0,Y 367.66,Z 513.999,A -85,B 0,C 180,E1 -12867.809,E2 -12867.809} C_VEL
LIN {X 0,Y 367.548,Z 514.605,A -85,B 0,C 180,E1 -12870,E2 -12870} C_VEL
LIN {X 0,Y 367.66,Z 514.044,A -85,B 0,C 180,E1 -12872.191,E2 -12872.191} C_VEL
LIN {X 0,Y 367.648,Z 512.387,A -85,B 0,C 180,E1 -12874.385,E2 -12874.385} C_VEL
LIN {X 0,Y 367.922,Z 509.487,A -85,B 0,C 180,E1 -12876.636,E2 -12876.636} C_VEL
LIN {X 0,Y 368.341,Z 505.549,A -85,B 0,C 180,E1 -12878.78,E2 -12878.78} C_VEL
LIN {X 0,Y 368.968,Z 500.207,A -85,B 0,C 180,E1 -12880.98,E2 -12880.98} C_VEL
LIN {X 0,Y 369.982,Z 493.388,A -85,B 0,C 180,E1 -12883.176,E2 -12883.176} C_VEL
LIN {X 0,Y 371.111,Z 484.878,A -85,B 0,C 180,E1 -12885.374,E2 -12885.374} C_VEL
LIN {X 0,Y 372.517,Z 475.814,A -85,B 0,C 180,E1 -12887.286,E2 -12887.286} C_VEL
LIN {X 0,Y 373.957,Z 466.57,A -85,B 0,C 180,E1 -12888.916,E2 -12888.916} C_VEL
LIN {X 0,Y 375.641,Z 454.922,A -85,B 0,C 180,E1 -12890.634,E2 -12890.634} C_VEL
LIN {X 0,Y 377.427,Z 442.373,A -85,B 0,C 180,E1 -12892.152,E2 -12892.152} C_VEL
LIN {X 0,Y 379.139,Z 428.866,A -85,B 0,C 180,E1 -12893.486,E2 -12893.486} C_VEL
LIN {X 0,Y 380.704,Z 414.852,A -85,B 0,C 180,E1 -12894.597,E2 -12894.597} C_VEL
LIN {X 0,Y 381.679,Z 404.013,A -85,B 0,C 180,E1 -12895.291,E2 -12895.291} C_VEL
LIN {X 0,Y 378.774,Z 392.979,A -85,B 0,C 180,E1 -12896.161,E2 -12896.161} C_VEL
LIN {X 0,Y 376.691,Z 388.159,A -85,B 0,C 180,E1 -12896.568,E2 -12896.568} C_VEL
LIN {X 0,Y 371.554,Z 381.158,A -85,B 0,C 180,E1 -12897.298,E2 -12897.298} C_VEL
LIN {X 0,Y 367.055,Z 375.674,A -85,B 0,C 180,E1 -12897.873,E2 -12897.873} C_VEL
LIN {X 0,Y 364.097,Z 371.131,A -85,B 0,C 180,E1 -12898.263,E2 -12898.263} C_VEL
LIN {X 0,Y 363.269,Z 369.477,A -85,B 0,C 180,E1 -12898.378,E2 -12898.378} C_VEL
LIN {X 0,Y 361.317,Z 364.744,A -85,B 0,C 180,E1 -12898.673,E2 -12898.673} C_VEL
LIN {X 0,Y 361.177,Z 363.902,A -85,B 0,C 180,E1 -12898.722,E2 -12898.722} C_VEL
LIN {X 0,Y 361.27,Z 361.456,A -85,B 0,C 180,E1 -12901.684,E2 -12901.684} C_VEL
LIN {X 0,Y 361.371,Z 359.426,A -85,B 0,C 180,E1 -12904.332,E2 -12904.332} C_VEL
LIN {X 0,Y 361.478,Z 357.311,A -85,B 0,C 180,E1 -12907.142,E2 -12907.142} C_VEL
LIN {X 0,Y 361.549,Z 356.076,A -85,B 0,C 180,E1 -12908.964,E2 -12908.964} C_VEL
LIN {X 0,Y 361.795,Z 356.039,A -85,B 0,C 180,E1 -12912.425,E2 -12912.425} C_VEL
LIN {X 0,Y 361.817,Z 356.042,A -85,B 0,C 180,E1 -12915.946,E2 -12915.946} C_VEL
LIN {X 0,Y 361.835,Z 356.04,A -85,B 0,C 180,E1 -12919.244,E2 -12919.244} C_VEL
LIN {X 0,Y 361.863,Z 356.034,A -85,B 0,C 180,E1 -12922.776,E2 -12922.776} C_VEL
LIN {X 0,Y 361.853,Z 356.03,A -85,B 0,C 180,E1 -12925.719,E2 -12925.719} C_VEL
LIN {X 0,Y 361.875,Z 356.035,A -85,B 0,C 180,E1 -12929.672,E2 -12929.672} C_VEL
LIN {X 0,Y 361.953,Z 356.01,A -85,B 0,C 180,E1 -12933.475,E2 -12933.475} C_VEL
LIN {X 0,Y 361.888,Z 356.03,A -85,B 0,C 180,E1 -12937.144,E2 -12937.144} C_VEL
LIN {X 0,Y 361.904,Z 356.016,A -85,B 0,C 180,E1 -12940.723,E2 -12940.723} C_VEL
LIN {X 0,Y 361.931,Z 356.026,A -85,B 0,C 180,E1 -12943.066,E2 -12943.066} C_VEL
LIN {X 0,Y 361.998,Z 355.997,A -85,B 0,C 180,E1 -12946.528,E2 -12946.528} C_VEL
LIN {X 0,Y 362.034,Z 356.014,A -85,B 0,C 180,E1 -12949.938,E2 -12949.938} C_VEL
LIN {X 0,Y 362.149,Z 355.998,A -85,B 0,C 180,E1 -12952.192,E2 -12952.192} C_VEL
LIN {X 0,Y 362.117,Z 356.005,A -85,B 0,C 180,E1 -12954.431,E2 -12954.431} C_VEL
LIN {X 0,Y 362.281,Z 355.983,A -85,B 0,C 180,E1 -12957.776,E2 -12957.776} C_VEL
LIN {X 0,Y 362.426,Z 355.968,A -85,B 0,C 180,E1 -12960,E2 -12960} C_VEL
LIN {X 0,Y 362.281,Z 355.983,A -85,B 0,C 180,E1 -12962.223,E2 -12962.223} C_VEL
LIN {X 0,Y 362.17,Z 355.998,A -85,B 0,C 180,E1 -12966.686,E2 -12966.686} C_VEL
LIN {X 0,Y 362.072,Z 356.009,A -85,B 0,C 180,E1 -12968.933,E2 -12968.933} C_VEL
LIN {X 0,Y 361.958,Z 356.02,A -85,B 0,C 180,E1 -12972.332,E2 -12972.332} C_VEL
LIN {X 0,Y 361.959,Z 356.021,A -85,B 0,C 180,E1 -12974.62,E2 -12974.62} C_VEL
LIN {X 0,Y 361.957,Z 356.021,A -85,B 0,C 180,E1 -12978.099,E2 -12978.099} C_VEL
LIN {X 0,Y 361.889,Z 356.035,A -85,B 0,C 180,E1 -12981.653,E2 -12981.653} C_VEL
LIN {X 0,Y 361.926,Z 356.029,A -85,B 0,C 180,E1 -12985.29,E2 -12985.29} C_VEL
LIN {X 0,Y 361.92,Z 356.032,A -85,B 0,C 180,E1 -12987.778,E2 -12987.778} C_VEL
LIN {X 0,Y 361.844,Z 356.039,A -85,B 0,C 180,E1 -12991.286,E2 -12991.286} C_VEL
LIN {X 0,Y 361.853,Z 356.038,A -85,B 0,C 180,E1 -12994.28,E2 -12994.28} C_VEL
LIN {X 0,Y 361.883,Z 356.112,A -85,B 0,C 180,E1 -12996.15,E2 -12996.15} C_VEL
LIN {X 0,Y 362.475,Z 359.558,A -85,B 0,C 180,E1 -12999.145,E2 -12999.145} C_VEL
LIN {X 0,Y 363.2,Z 363.98,A -85,B 0,C 180,E1 -13002.668,E2 -13002.668} C_VEL
LIN {X 0,Y 363.952,Z 368.424,A -85,B 0,C 180,E1 -13005.96,E2 -13005.96} C_VEL
LIN {X 0,Y 364.174,Z 370.66,A -85,B 0,C 180,E1 -13007.512,E2 -13007.512} C_VEL
LIN {X 0,Y 363.981,Z 373.978,A -85,B 0,C 180,E1 -13009.697,E2 -13009.697} C_VEL
LIN {X 0,Y 363.375,Z 379.52,A -85,B 0,C 180,E1 -13013.162,E2 -13013.162} C_VEL
LIN {X 0,Y 362.827,Z 384.864,A -85,B 0,C 180,E1 -13016.399,E2 -13016.399} C_VEL
LIN {X 0,Y 362.277,Z 390.44,A -85,B 0,C 180,E1 -13019.71,E2 -13019.71} C_VEL
LIN {X 0,Y 361.956,Z 393.232,A -85,B 0,C 180,E1 -13021.351,E2 -13021.351} C_VEL
LIN {X 0,Y 363.797,Z 399.612,A -85,B 0,C 180,E1 -13021.68,E2 -13021.68} C_VEL
LIN {X 0,Y 367.828,Z 413.761,A -85,B 0,C 180,E1 -13022.485,E2 -13022.485} C_VEL
LIN {X 0,Y 370.957,Z 428.117,A -85,B 0,C 180,E1 -13023.414,E2 -13023.414} C_VEL
LIN {X 0,Y 373.246,Z 442.553,A -85,B 0,C 180,E1 -13024.49,E2 -13024.49} C_VEL
LIN {X 0,Y 373.219,Z 446.894,A -85,B 0,C 180,E1 -13024.81,E2 -13024.81} C_VEL
LIN {X 0,Y 371.571,Z 460.464,A -85,B 0,C 180,E1 -13025.857,E2 -13025.857} C_VEL
LIN {X 0,Y 369.789,Z 473.231,A -85,B 0,C 180,E1 -13027.07,E2 -13027.07} C_VEL
LIN {X 0,Y 367.814,Z 486.153,A -85,B 0,C 180,E1 -13028.566,E2 -13028.566} C_VEL
LIN {X 0,Y 366.155,Z 497.33,A -85,B 0,C 180,E1 -13030.137,E2 -13030.137} C_VEL
LIN {X 0,Y 364.774,Z 507.026,A -85,B 0,C 180,E1 -13031.755,E2 -13031.755} C_VEL
LIN {X 0,Y 363.431,Z 515.581,A -85,B 0,C 180,E1 -13033.428,E2 -13033.428} C_VEL
LIN {X 0,Y 362.316,Z 523.969,A -85,B 0,C 180,E1 -13035.395,E2 -13035.395} C_VEL
LIN {X 0,Y 361.394,Z 531.86,A -85,B 0,C 180,E1 -13037.649,E2 -13037.649} C_VEL
LIN {X 0,Y 360.745,Z 538.145,A -85,B 0,C 180,E1 -13039.902,E2 -13039.902} C_VEL
LIN {X 0,Y 360.492,Z 543.018,A -85,B 0,C 180,E1 -13042.157,E2 -13042.157} C_VEL
LIN {X 0,Y 360.361,Z 546.591,A -85,B 0,C 180,E1 -13044.404,E2 -13044.404} C_VEL
LIN {X 0,Y 360.327,Z 548.943,A -85,B 0,C 180,E1 -13046.646,E2 -13046.646} C_VEL
LIN {X 0,Y 360.47,Z 550.134,A -85,B 0,C 180,E1 -13048.883,E2 -13048.883} C_VEL
LIN {X 0,Y 360.47,Z 550.132,A -85,B 0,C 180,E1 -13051.118,E2 -13051.118} C_VEL
LIN {X 0,Y 360.329,Z 548.933,A -85,B 0,C 180,E1 -13053.355,E2 -13053.355} C_VEL
LIN {X 0,Y 360.415,Z 546.577,A -85,B 0,C 180,E1 -13055.596,E2 -13055.596} C_VEL
LIN {X 0,Y 360.494,Z 543.001,A -85,B 0,C 180,E1 -13057.844,E2 -13057.844} C_VEL
LIN {X 0,Y 360.746,Z 538.123,A -85,B 0,C 180,E1 -13060.099,E2 -13060.099} C_VEL
LIN {X 0,Y 361.399,Z 531.824,A -85,B 0,C 180,E1 -13062.352,E2 -13062.352} C_VEL
LIN {X 0,Y 362.317,Z 523.922,A -85,B 0,C 180,E1 -13064.606,E2 -13064.606} C_VEL
LIN {X 0,Y 363.434,Z 515.528,A -85,B 0,C 180,E1 -13066.573,E2 -13066.573} C_VEL
LIN {X 0,Y 364.988,Z 505.435,A -85,B 0,C 180,E1 -13068.525,E2 -13068.525} C_VEL
LIN {X 0,Y 366.516,Z 495.12,A -85,B 0,C 180,E1 -13070.192,E2 -13070.192} C_VEL
LIN {X 0,Y 368.367,Z 482.842,A -85,B 0,C 180,E1 -13071.842,E2 -13071.842} C_VEL
LIN {X 0,Y 370.127,Z 470.529,A -85,B 0,C 180,E1 -13073.204,E2 -13073.204} C_VEL
LIN {X 0,Y 372.01,Z 457.145,A -85,B 0,C 180,E1 -13074.41,E2 -13074.41} C_VEL
LIN {X 0,Y 373.378,Z 444.033,A -85,B 0,C 180,E1 -13075.379,E2 -13075.379} C_VEL
LIN {X 0,Y 371.268,Z 429.805,A -85,B 0,C 180,E1 -13076.454,E2 -13076.454} C_VEL
LIN {X 0,Y 367.897,Z 414.005,A -85,B 0,C 180,E1 -13077.486,E2 -13077.486} C_VEL
LIN {X 0,Y 363.768,Z 399.507,A -85,B 0,C 180,E1 -13078.31,E2 -13078.31} C_VEL
LIN {X 0,Y 362.011,Z 393.664,A -85,B 0,C 180,E1 -13078.604,E2 -13078.604} C_VEL
LIN {X 0,Y 361.965,Z 393.204,A -85,B 0,C 180,E1 -13078.652,E2 -13078.652} C_VEL
LIN {X 0,Y 362.428,Z 388.261,A -85,B 0,C 180,E1 -13081.572,E2 -13081.572} C_VEL
LIN {X 0,Y 363.039,Z 382.759,A -85,B 0,C 180,E1 -13084.826,E2 -13084.826} C_VEL
LIN {X 0,Y 363.59,Z 377.274,A -85,B 0,C 180,E1 -13088.21,E2 -13088.21} C_VEL
LIN {X 0,Y 364.113,Z 372.577,A -85,B 0,C 180,E1 -13091.17,E2 -13091.17} C_VEL
LIN {X 0,Y 364.103,Z 370.069,A -85,B 0,C 180,E1 -13092.821,E2 -13092.821} C_VEL
LIN {X 0,Y 363.549,Z 365.789,A -85,B 0,C 180,E1 -13095.898,E2 -13095.898} C_VEL
LIN {X 0,Y 362.842,Z 361.657,A -85,B 0,C 180,E1 -13099.061,E2 -13099.061} C_VEL
LIN {X 0,Y 362.11,Z 357.336,A -85,B 0,C 180,E1 -13102.727,E2 -13102.727} C_VEL
LIN {X 0,Y 361.889,Z 356.037,A -85,B 0,C 180,E1 -13104.023,E2 -13104.023} C_VEL
LIN {X 0,Y 361.85,Z 356.039,A -85,B 0,C 180,E1 -13107.056,E2 -13107.056} C_VEL
LIN {X 0,Y 361.903,Z 356.032,A -85,B 0,C 180,E1 -13110.956,E2 -13110.956} C_VEL
LIN {X 0,Y 361.956,Z 356.025,A -85,B 0,C 180,E1 -13113.475,E2 -13113.475} C_VEL
LIN {X 0,Y 361.893,Z 356.033,A -85,B 0,C 180,E1 -13117.145,E2 -13117.145} C_VEL
LIN {X 0,Y 361.924,Z 356.027,A -85,B 0,C 180,E1 -13120.724,E2 -13120.724} C_VEL
LIN {X 0,Y 361.949,Z 356.027,A -85,B 0,C 180,E1 -13124.226,E2 -13124.226} C_VEL
LIN {X 0,Y 362.002,Z 356.021,A -85,B 0,C 180,E1 -13126.528,E2 -13126.528} C_VEL
LIN {X 0,Y 362.035,Z 356.016,A -85,B 0,C 180,E1 -13129.938,E2 -13129.938} C_VEL
LIN {X 0,Y 362.155,Z 356.004,A -85,B 0,C 180,E1 -13132.193,E2 -13132.193} C_VEL
LIN {X 0,Y 362.121,Z 356.003,A -85,B 0,C 180,E1 -13134.431,E2 -13134.431} C_VEL
LIN {X 0,Y 362.286,Z 355.982,A -85,B 0,C 180,E1 -13137.777,E2 -13137.777} C_VEL
LIN {X 0,Y 362.43,Z 355.963,A -85,B 0,C 180,E1 -13140,E2 -13140} C_VEL
LIN {X 0,Y 362.286,Z 355.982,A -85,B 0,C 180,E1 -13142.224,E2 -13142.224} C_VEL
LIN {X 0,Y 362.176,Z 355.991,A -85,B 0,C 180,E1 -13146.686,E2 -13146.686} C_VEL
LIN {X 0,Y 362.078,Z 356.011,A -85,B 0,C 180,E1 -13148.933,E2 -13148.933} C_VEL
LIN {X 0,Y 361.963,Z 355.998,A -85,B 0,C 180,E1 -13152.332,E2 -13152.332} C_VEL
LIN {X 0,Y 361.965,Z 356.012,A -85,B 0,C 180,E1 -13154.62,E2 -13154.62} C_VEL
LIN {X 0,Y 361.959,Z 356.018,A -85,B 0,C 180,E1 -13158.099,E2 -13158.099} C_VEL
LIN {X 0,Y 361.884,Z 356.019,A -85,B 0,C 180,E1 -13161.654,E2 -13161.654} C_VEL
LIN {X 0,Y 361.93,Z 356.024,A -85,B 0,C 180,E1 -13165.29,E2 -13165.29} C_VEL
LIN {X 0,Y 361.911,Z 356.013,A -85,B 0,C 180,E1 -13167.779,E2 -13167.779} C_VEL
LIN {X 0,Y 361.841,Z 356.035,A -85,B 0,C 180,E1 -13171.629,E2 -13171.629} C_VEL
LIN {X 0,Y 361.878,Z 356.033,A -85,B 0,C 180,E1 -13175.345,E2 -13175.345} C_VEL
LIN {X 0,Y 361.874,Z 356.035,A -85,B 0,C 180,E1 -13179.027,E2 -13179.027} C_VEL
LIN {X 0,Y 361.839,Z 356.04,A -85,B 0,C 180,E1 -13182.829,E2 -13182.829} C_VEL
LIN {X 0,Y 361.811,Z 356.046,A -85,B 0,C 180,E1 -13185.948,E2 -13185.948} C_VEL
LIN {X 0,Y 361.741,Z 356.056,A -85,B 0,C 180,E1 -13188.657,E2 -13188.657} C_VEL
LIN {X 0,Y 361.491,Z 356.259,A -85,B 0,C 180,E1 -13191.527,E2 -13191.527} C_VEL
LIN {X 0,Y 361.406,Z 358.625,A -85,B 0,C 180,E1 -13194.76,E2 -13194.76} C_VEL
LIN {X 0,Y 361.384,Z 360.326,A -85,B 0,C 180,E1 -13197.007,E2 -13197.007} C_VEL
LIN {X 0,Y 361.201,Z 363.516,A -85,B 0,C 180,E1 -13200.893,E2 -13200.893} C_VEL
LIN {X 0,Y 361.209,Z 363.938,A -85,B 0,C 180,E1 -13201.389,E2 -13201.389} C_VEL
LIN {X 0,Y 362.28,Z 367.106,A -85,B 0,C 180,E1 -13201.58,E2 -13201.58} C_VEL
LIN {X 0,Y 368.181,Z 381.859,A -85,B 0,C 180,E1 -13202.576,E2 -13202.576} C_VEL
LIN {X 0,Y 372.202,Z 394.277,A -85,B 0,C 180,E1 -13203.494,E2 -13203.494} C_VEL
LIN {X 0,Y 375.048,Z 404.809,A -85,B 0,C 180,E1 -13204.362,E2 -13204.362} C_VEL
LIN {X 0,Y 373.994,Z 417.722,A -85,B 0,C 180,E1 -13205.244,E2 -13205.244} C_VEL
LIN {X 0,Y 372.421,Z 431.084,A -85,B 0,C 180,E1 -13206.358,E2 -13206.358} C_VEL
LIN {X 0,Y 370.591,Z 444.251,A -85,B 0,C 180,E1 -13207.71,E2 -13207.71} C_VEL
LIN {X 0,Y 368.949,Z 455.671,A -85,B 0,C 180,E1 -13209.136,E2 -13209.136} C_VEL
LIN {X 0,Y 367.301,Z 466.332,A -85,B 0,C 180,E1 -13210.727,E2 -13210.727} C_VEL
LIN {X 0,Y 365.58,Z 477.083,A -85,B 0,C 180,E1 -13212.663,E2 -13212.663} C_VEL
LIN {X 0,Y 364.128,Z 486.071,A -85,B 0,C 180,E1 -13214.627,E2 -13214.627} C_VEL
LIN {X 0,Y 363.126,Z 493.372,A -85,B 0,C 180,E1 -13216.57,E2 -13216.57} C_VEL
LIN {X 0,Y 362.207,Z 498.684,A -85,B 0,C 180,E1 -13218.244,E2 -13218.244} C_VEL
LIN {X 0,Y 361.49,Z 504.461,A -85,B 0,C 180,E1 -13220.488,E2 -13220.488} C_VEL
LIN {X 0,Y 361.058,Z 507.881,A -85,B 0,C 180,E1 -13222.168,E2 -13222.168} C_VEL
LIN {X 0,Y 360.742,Z 511.341,A -85,B 0,C 180,E1 -13224.409,E2 -13224.409} C_VEL
LIN {X 0,Y 360.558,Z 513.628,A -85,B 0,C 180,E1 -13226.647,E2 -13226.647} C_VEL
LIN {X 0,Y 360.521,Z 514.794,A -85,B 0,C 180,E1 -13228.883,E2 -13228.883} C_VEL
LIN {X 0,Y 360.521,Z 514.808,A -85,B 0,C 180,E1 -13231.117,E2 -13231.117} C_VEL
LIN {X 0,Y 360.557,Z 513.703,A -85,B 0,C 180,E1 -13233.352,E2 -13233.352} C_VEL
LIN {X 0,Y 360.741,Z 511.474,A -85,B 0,C 180,E1 -13235.59,E2 -13235.59} C_VEL
LIN {X 0,Y 361.049,Z 508.068,A -85,B 0,C 180,E1 -13237.831,E2 -13237.831} C_VEL
LIN {X 0,Y 361.621,Z 503.398,A -85,B 0,C 180,E1 -13240.073,E2 -13240.073} C_VEL
LIN {X 0,Y 362.39,Z 497.346,A -85,B 0,C 180,E1 -13242.317,E2 -13242.317} C_VEL
LIN {X 0,Y 363.442,Z 490.756,A -85,B 0,C 180,E1 -13244.273,E2 -13244.273} C_VEL
LIN {X 0,Y 364.614,Z 482.793,A -85,B 0,C 180,E1 -13246.229,E2 -13246.229} C_VEL
LIN {X 0,Y 366.207,Z 473.221,A -85,B 0,C 180,E1 -13248.171,E2 -13248.171} C_VEL
LIN {X 0,Y 367.722,Z 463.431,A -85,B 0,C 180,E1 -13249.83,E2 -13249.83} C_VEL
LIN {X 0,Y 369.546,Z 451.774,A -85,B 0,C 180,E1 -13251.474,E2 -13251.474} C_VEL
LIN {X 0,Y 371.247,Z 440.161,A -85,B 0,C 180,E1 -13252.835,E2 -13252.835} C_VEL
LIN {X 0,Y 372.827,Z 427.637,A -85,B 0,C 180,E1 -13254.056,E2 -13254.056} C_VEL
LIN {X 0,Y 374.391,Z 414.147,A -85,B 0,C 180,E1 -13255.119,E2 -13255.119} C_VEL
LIN {X 0,Y 375.03,Z 404.654,A -85,B 0,C 180,E1 -13255.752,E2 -13255.752} C_VEL
LIN {X 0,Y 370.857,Z 389.774,A -85,B 0,C 180,E1 -13256.946,E2 -13256.946} C_VEL
LIN {X 0,Y 365.945,Z 375.975,A -85,B 0,C 180,E1 -13257.94,E2 -13257.94} C_VEL
LIN {X 0,Y 363.269,Z 369.477,A -85,B 0,C 180,E1 -13258.378,E2 -13258.378} C_VEL
LIN {X 0,Y 361.699,Z 366.799,A -85,B 0,C 180,E1 -13258.69,E2 -13258.69} C_VEL
LIN {X 0,Y 360.067,Z 364.993,A -85,B 0,C 180,E1 -13259.14,E2 -13259.14} C_VEL
LIN {X 0,Y 357.809,Z 363.448,A -85,B 0,C 180,E1 -13259.963,E2 -13259.963} C_VEL
LIN {X 0,Y 355.055,Z 362.346,A -85,B 0,C 180,E1 -13261.593,E2 -13261.593} C_VEL
LIN {X 0,Y 354.282,Z 361.372,A -85,B 0,C 180,E1 -13262.97,E2 -13262.97} C_VEL
LIN {X 0,Y 354.389,Z 358.746,A -85,B 0,C 180,E1 -13266.508,E2 -13266.508} C_VEL
LIN {X 0,Y 354.547,Z 356.947,A -85,B 0,C 180,E1 -13269.369,E2 -13269.369} C_VEL
LIN {X 0,Y 354.76,Z 356.917,A -85,B 0,C 180,E1 -13272.862,E2 -13272.862} C_VEL
LIN {X 0,Y 354.766,Z 356.921,A -85,B 0,C 180,E1 -13276.103,E2 -13276.103} C_VEL
LIN {X 0,Y 354.787,Z 356.918,A -85,B 0,C 180,E1 -13279.179,E2 -13279.179} C_VEL
LIN {X 0,Y 354.807,Z 356.915,A -85,B 0,C 180,E1 -13282.402,E2 -13282.402} C_VEL
LIN {X 0,Y 354.811,Z 356.914,A -85,B 0,C 180,E1 -13284.941,E2 -13284.941} C_VEL
